// TIA Portal V20 export
FUNCTION_BLOCK "Sequence_2_AlignTable"   // FB243, LAD
AUTHOR : ERsystem_FA2_DH. Kim
// stored: IsIECCheckEnabled true, MemoryReserve 100, Namespace Unit1.Em4, SetENOAutomatically false
   VAR
      instSequenceLADStatus { ExternalWritable := 'False'} : "LAF_StatusLadSequence";
      instSequenceLADControl { ExternalWritable := 'False'} : "LAF_ControlLadSequence";
      statTonTime { ExternalWritable := 'False'} : Array[0..9999] of TON_TIME;
   END_VAR
   VAR_TEMP
      tempCustomerAction : Bool;   // Placeholder for possible actions
      tempDo_nothing_and_wait_for_init : Bool;   // Placeholder for doing nothing
      tempSafeStateCondition : Bool;   // Temp Condition for the equipment module to be in a safe state
   END_VAR
   VAR CONSTANT
      delayTime : Time := T#300ms;
      STEP_IDLE : DInt := 1;
      STEP_IMMEDIATE_STOP : DInt := 9001;   // Step executed when an immediate stop command is triggered for the sequence (i.e. when unit is in state aborting)
      JOB_1_STEP_01 : DInt := 101;
      JOB_1_STEP_10 : DInt := 110;
      JOB_1_STEP_20 : DInt := 120;
      JOB_1_STEP_30 : DInt := 130;
      JOB_1_STEP_40 : DInt := 140;
      JOB_1_STEP_41 : DInt := 141;
      JOB_1_STEP_42 : DInt := 142;
      JOB_1_STEP_50 : DInt := 150;
      JOB_1_STEP_51 : DInt := 151;
      JOB_1_STEP_52 : DInt := 152;
      JOB_1_STEP_60 : DInt := 160;
      JOB_1_STEP_61 : DInt := 161;
      JOB_1_STEP_62 : DInt := 162;
      JOB_1_STEP_70 : DInt := 170;
      JOB_1_STEP_80 : DInt := 180;
      JOB_1_STEP_81 : DInt := 181;
      JOB_1_STEP_90 : DInt := 190;
      JOB_2_STEP_01 : DInt := 201;
      JOB_2_STEP_10 : DInt := 210;
      JOB_2_STEP_20 : DInt := 220;
      JOB_2_STEP_30 : DInt := 230;
      JOB_2_STEP_90 : DInt := 290;
      JOB_3_STEP_01 : DInt := 301;
      JOB_3_STEP_10 : DInt := 310;
      JOB_3_STEP_20 : DInt := 320;
      JOB_3_STEP_80 : DInt := 380;
      JOB_3_STEP_90 : DInt := 390;
      JOB_4_STEP_01 : DInt := 401;
      JOB_4_STEP_10 : DInt := 410;
      JOB_4_STEP_11 : DInt := 411;
      JOB_4_STEP_20 : DInt := 420;
      JOB_4_STEP_21 : DInt := 421;
      JOB_4_STEP_30 : DInt := 430;
      JOB_4_STEP_80 : DInt := 480;
      JOB_4_STEP_81 : DInt := 481;
      JOB_4_STEP_90 : DInt := 490;
      JOB_22_STEP_01 : DInt := 2201;
      JOB_22_STEP_10 : DInt := 2210;
      JOB_22_STEP_20 : DInt := 2220;
      JOB_22_STEP_30 : DInt := 2230;
      JOB_22_STEP_40 : DInt := 2240;
      JOB_22_STEP_50 : DInt := 2250;
      JOB_22_STEP_80 : DInt := 2280;
      JOB_22_STEP_81 : DInt := 2281;
      JOB_22_STEP_90 : DInt := 2290;
      FALSE : Bool := FALSE;
      TRUE : Bool := TRUE;
   END_VAR
   VAR_TEMP   // added for the SCL form of the ladder/FBD networks
      _w1 : Bool;
   END_VAR
BEGIN

REGION Network 1: BLOCK INFO HEADER
   // (company) / (C) Copyright (year)
   // ---------------------------------------------------------------------------------
   // Title:                             (Title of this block)
   // Comment/Function: (that is implemented in the block)
   // Library/Family:           (that the source is dedicated to)
   // Author:                        (department / person in charge / contact)
   // Target System:          (test system with FW version)
   // Engineering:              TIA Portal (SW version)
   // Restrictions:               (OB types, etc.)
   // Requirements:           (hardware, technological package, etc.)
   // ---------------------------------------------------------------------------------
   // Change log table:
   // Version          | Date             | Signature      | Expert in charge  | Changes applied ------------------------|----------------------|-------------------------|--------------------------------|-----------------------
   // 001.000.000 | yyyy-mm-dd | 0x00000000 | (name of expert) | First released version
END_REGION

REGION Network 2: DESCRIPTION
   // This is a template block provided by the Automation Framework. It can be used to create an own project.
   // The Block Info Header is prepared to put in your own data.
   // Description of the block could be added here and the docu created by Code2Docu.
END_REGION

REGION Network 3: ******************** CONTROL ********************
END_REGION

REGION Network 4: Sequence Control
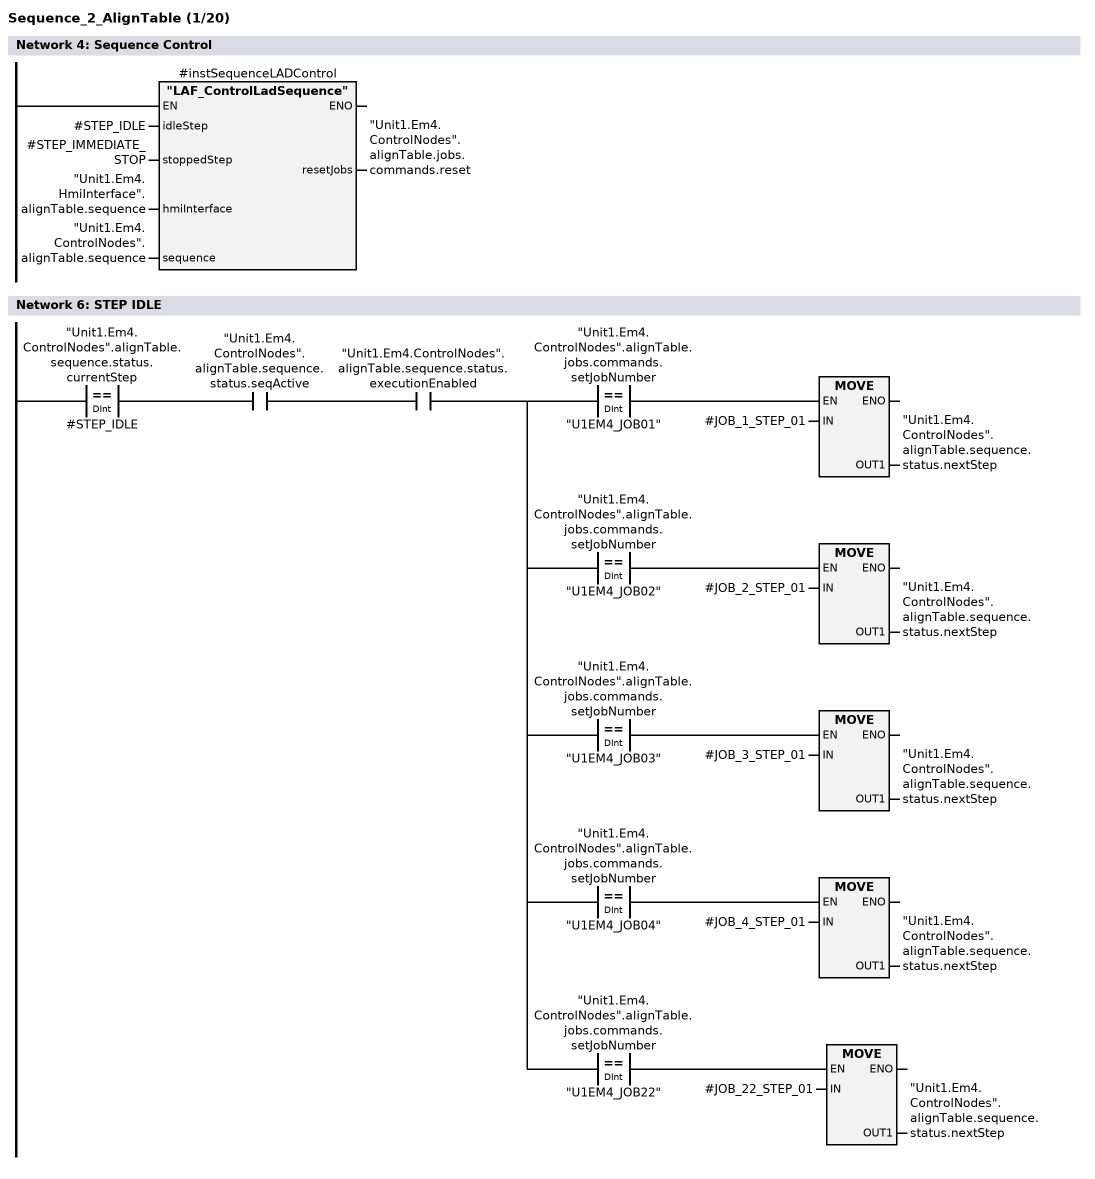
   RUNG wire#powerrail
      #instSequenceLADControl(idleStep := #STEP_IDLE, stoppedStep := #STEP_IMMEDIATE_STOP, hmiInterface := "Unit1.Em4.HmiInterface".alignTable.sequence, sequence := "Unit1.Em4.ControlNodes".alignTable.sequence, resetJobs => "Unit1.Em4.ControlNodes".alignTable.jobs.commands.reset)
   END_RUNG
   // the same network as SCL:
   #instSequenceLADControl(idleStep := #STEP_IDLE,   // "LAF_ControlLadSequence"
                           stoppedStep := #STEP_IMMEDIATE_STOP,
                           hmiInterface := "Unit1.Em4.HmiInterface".alignTable.sequence,
                           sequence := "Unit1.Em4.ControlNodes".alignTable.sequence,
                           resetJobs => "Unit1.Em4.ControlNodes".alignTable.jobs.commands.reset);
END_REGION

REGION Network 5: ******************** JOB SELECT ********************
END_REGION

REGION Network 6: STEP IDLE
   RUNG wire#powerrail
      { S7_Templates := "SrcType := DInt" } EQ_Contact(in1 := "Unit1.Em4.ControlNodes".alignTable.sequence.status.currentStep, in2 := #STEP_IDLE)
      Contact( "Unit1.Em4.ControlNodes".alignTable.sequence.status.seqActive )
      Contact( "Unit1.Em4.ControlNodes".alignTable.sequence.status.executionEnabled )
      wire#w1
      { S7_Templates := "SrcType := DInt" } EQ_Contact(in1 := "Unit1.Em4.ControlNodes".alignTable.jobs.commands.setJobNumber, in2 := "U1EM4_JOB01")
      Move(in := #JOB_1_STEP_01, out1 => "Unit1.Em4.ControlNodes".alignTable.sequence.status.nextStep)
   END_RUNG
   RUNG wire#w1
      { S7_Templates := "SrcType := DInt" } EQ_Contact(in1 := "Unit1.Em4.ControlNodes".alignTable.jobs.commands.setJobNumber, in2 := "U1EM4_JOB02")
      Move(in := #JOB_2_STEP_01, out1 => "Unit1.Em4.ControlNodes".alignTable.sequence.status.nextStep)
   END_RUNG
   RUNG wire#w1
      { S7_Templates := "SrcType := DInt" } EQ_Contact(in1 := "Unit1.Em4.ControlNodes".alignTable.jobs.commands.setJobNumber, in2 := "U1EM4_JOB03")
      Move(in := #JOB_3_STEP_01, out1 => "Unit1.Em4.ControlNodes".alignTable.sequence.status.nextStep)
   END_RUNG
   RUNG wire#w1
      { S7_Templates := "SrcType := DInt" } EQ_Contact(in1 := "Unit1.Em4.ControlNodes".alignTable.jobs.commands.setJobNumber, in2 := "U1EM4_JOB04")
      Move(in := #JOB_4_STEP_01, out1 => "Unit1.Em4.ControlNodes".alignTable.sequence.status.nextStep)
   END_RUNG
   RUNG wire#w1
      { S7_Templates := "SrcType := DInt" } EQ_Contact(in1 := "Unit1.Em4.ControlNodes".alignTable.jobs.commands.setJobNumber, in2 := "U1EM4_JOB22")
      Move(in := #JOB_22_STEP_01, out1 => "Unit1.Em4.ControlNodes".alignTable.sequence.status.nextStep)
   END_RUNG
   // the same network as SCL:
   #_w1 := ("Unit1.Em4.ControlNodes".alignTable.sequence.status.currentStep = #STEP_IDLE) AND "Unit1.Em4.ControlNodes".alignTable.sequence.status.seqActive AND "Unit1.Em4.ControlNodes".alignTable.sequence.status.executionEnabled;
   IF #_w1 AND ("Unit1.Em4.ControlNodes".alignTable.jobs.commands.setJobNumber = "U1EM4_JOB01") THEN
       "Unit1.Em4.ControlNodes".alignTable.sequence.status.nextStep := #JOB_1_STEP_01;
   END_IF;
   IF #_w1 AND ("Unit1.Em4.ControlNodes".alignTable.jobs.commands.setJobNumber = "U1EM4_JOB02") THEN
       "Unit1.Em4.ControlNodes".alignTable.sequence.status.nextStep := #JOB_2_STEP_01;
   END_IF;
   IF #_w1 AND ("Unit1.Em4.ControlNodes".alignTable.jobs.commands.setJobNumber = "U1EM4_JOB03") THEN
       "Unit1.Em4.ControlNodes".alignTable.sequence.status.nextStep := #JOB_3_STEP_01;
   END_IF;
   IF #_w1 AND ("Unit1.Em4.ControlNodes".alignTable.jobs.commands.setJobNumber = "U1EM4_JOB04") THEN
       "Unit1.Em4.ControlNodes".alignTable.sequence.status.nextStep := #JOB_4_STEP_01;
   END_IF;
   IF #_w1 AND ("Unit1.Em4.ControlNodes".alignTable.jobs.commands.setJobNumber = "U1EM4_JOB22") THEN
       "Unit1.Em4.ControlNodes".alignTable.sequence.status.nextStep := #JOB_22_STEP_01;
   END_IF;
END_REGION

REGION Network 7: ******************** JOB[1] EM HOMING ********************
END_REGION

REGION Network 8: Step[101] : JOB[1] Condition
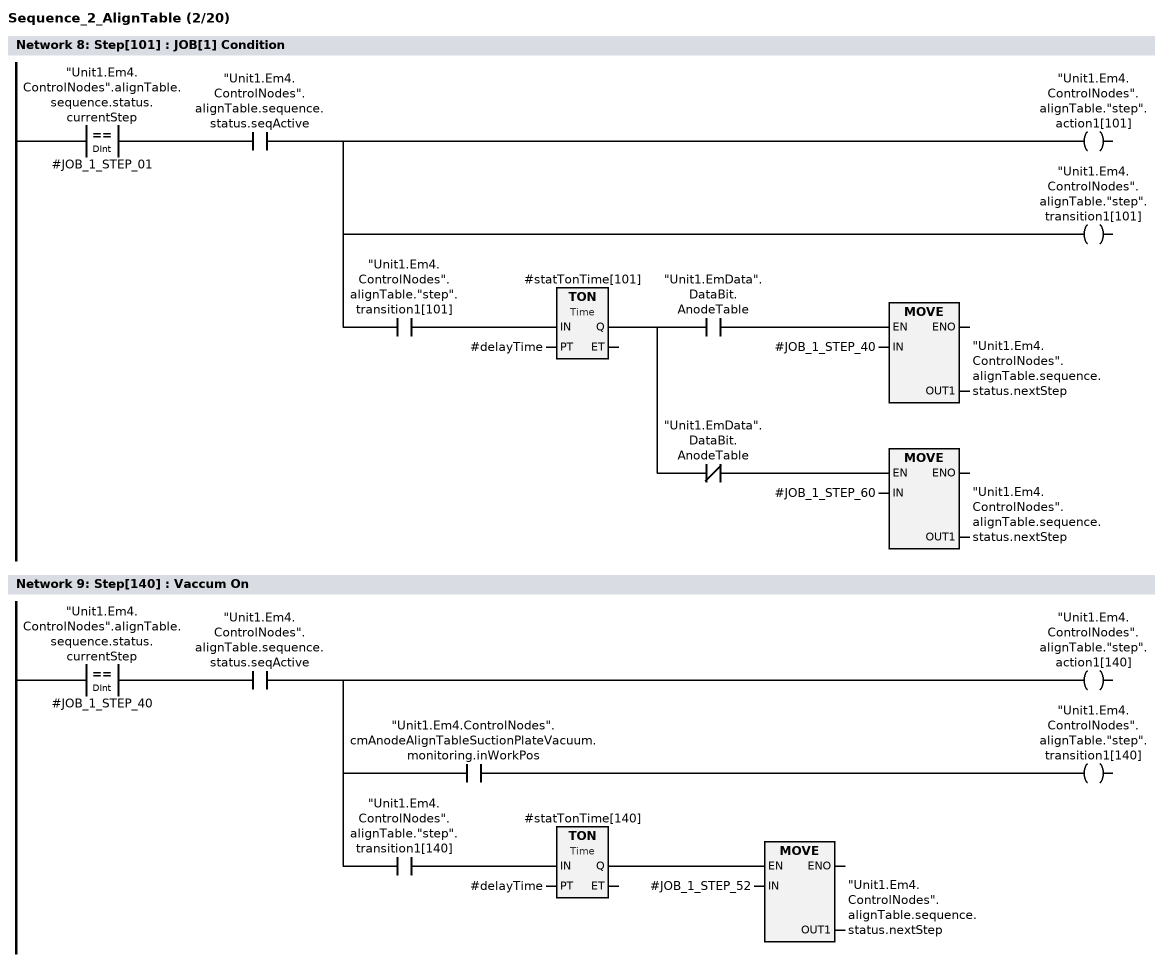
   RUNG wire#powerrail
      { S7_Templates := "SrcType := DInt" } EQ_Contact(in1 := "Unit1.Em4.ControlNodes".alignTable.sequence.status.currentStep, in2 := #JOB_1_STEP_01)
      Contact( "Unit1.Em4.ControlNodes".alignTable.sequence.status.seqActive )
      wire#w1
      Coil( "Unit1.Em4.ControlNodes".alignTable."step".action1[101] )
   END_RUNG
   RUNG wire#w1
      Coil( "Unit1.Em4.ControlNodes".alignTable."step".transition1[101] )
   END_RUNG
   RUNG wire#w1
      Contact( "Unit1.Em4.ControlNodes".alignTable."step".transition1[101] )
      { S7_Templates := "time_type := Time" } #statTonTime[101].TON(pt := #delayTime, et =>)
      wire#w2
      Contact( "Unit1.EmData".DataBit.AnodeTable )
      Move(in := #JOB_1_STEP_40, out1 => "Unit1.Em4.ControlNodes".alignTable.sequence.status.nextStep)
   END_RUNG
   RUNG wire#w2
      I_Contact( "Unit1.EmData".DataBit.AnodeTable )
      Move(in := #JOB_1_STEP_60, out1 => "Unit1.Em4.ControlNodes".alignTable.sequence.status.nextStep)
   END_RUNG
   // the same network as SCL:
   "Unit1.Em4.ControlNodes".alignTable."step".action1[101] := ("Unit1.Em4.ControlNodes".alignTable.sequence.status.currentStep = #JOB_1_STEP_01) AND "Unit1.Em4.ControlNodes".alignTable.sequence.status.seqActive;
   "Unit1.Em4.ControlNodes".alignTable."step".transition1[101] := ("Unit1.Em4.ControlNodes".alignTable.sequence.status.currentStep = #JOB_1_STEP_01) AND "Unit1.Em4.ControlNodes".alignTable.sequence.status.seqActive;
   #statTonTime[101].TON(IN := ("Unit1.Em4.ControlNodes".alignTable.sequence.status.currentStep = #JOB_1_STEP_01) AND "Unit1.Em4.ControlNodes".alignTable.sequence.status.seqActive AND "Unit1.Em4.ControlNodes".alignTable."step".transition1[101],
                         PT := #delayTime);
   IF #statTonTime[101].Q AND "Unit1.EmData".DataBit.AnodeTable THEN
       "Unit1.Em4.ControlNodes".alignTable.sequence.status.nextStep := #JOB_1_STEP_40;
   END_IF;
   IF #statTonTime[101].Q AND NOT "Unit1.EmData".DataBit.AnodeTable THEN
       "Unit1.Em4.ControlNodes".alignTable.sequence.status.nextStep := #JOB_1_STEP_60;
   END_IF;
END_REGION

REGION Network 9: Step[140] : Vaccum On
   RUNG wire#powerrail
      { S7_Templates := "SrcType := DInt" } EQ_Contact(in1 := "Unit1.Em4.ControlNodes".alignTable.sequence.status.currentStep, in2 := #JOB_1_STEP_40)
      Contact( "Unit1.Em4.ControlNodes".alignTable.sequence.status.seqActive )
      wire#w1
      Coil( "Unit1.Em4.ControlNodes".alignTable."step".action1[140] )
   END_RUNG
   RUNG wire#w1
      Contact( "Unit1.Em4.ControlNodes".cmAnodeAlignTableSuctionPlateVacuum.monitoring.inWorkPos )
      Coil( "Unit1.Em4.ControlNodes".alignTable."step".transition1[140] )
   END_RUNG
   RUNG wire#w1
      Contact( "Unit1.Em4.ControlNodes".alignTable."step".transition1[140] )
      { S7_Templates := "time_type := Time" } #statTonTime[140].TON(pt := #delayTime, et =>)
      Move(in := #JOB_1_STEP_52, out1 => "Unit1.Em4.ControlNodes".alignTable.sequence.status.nextStep)
   END_RUNG
   // the same network as SCL:
   "Unit1.Em4.ControlNodes".alignTable."step".action1[140] := ("Unit1.Em4.ControlNodes".alignTable.sequence.status.currentStep = #JOB_1_STEP_40) AND "Unit1.Em4.ControlNodes".alignTable.sequence.status.seqActive;
   "Unit1.Em4.ControlNodes".alignTable."step".transition1[140] := ("Unit1.Em4.ControlNodes".alignTable.sequence.status.currentStep = #JOB_1_STEP_40) AND "Unit1.Em4.ControlNodes".alignTable.sequence.status.seqActive AND "Unit1.Em4.ControlNodes".cmAnodeAlignTableSuctionPlateVacuum.monitoring.inWorkPos;
   #statTonTime[140].TON(IN := ("Unit1.Em4.ControlNodes".alignTable.sequence.status.currentStep = #JOB_1_STEP_40) AND "Unit1.Em4.ControlNodes".alignTable.sequence.status.seqActive AND "Unit1.Em4.ControlNodes".alignTable."step".transition1[140],
                         PT := #delayTime);
   IF #statTonTime[140].Q THEN
       "Unit1.Em4.ControlNodes".alignTable.sequence.status.nextStep := #JOB_1_STEP_52;
   END_IF;
END_REGION

REGION Network 10: Step[141] : Align Table → Main P&P [Load Done]
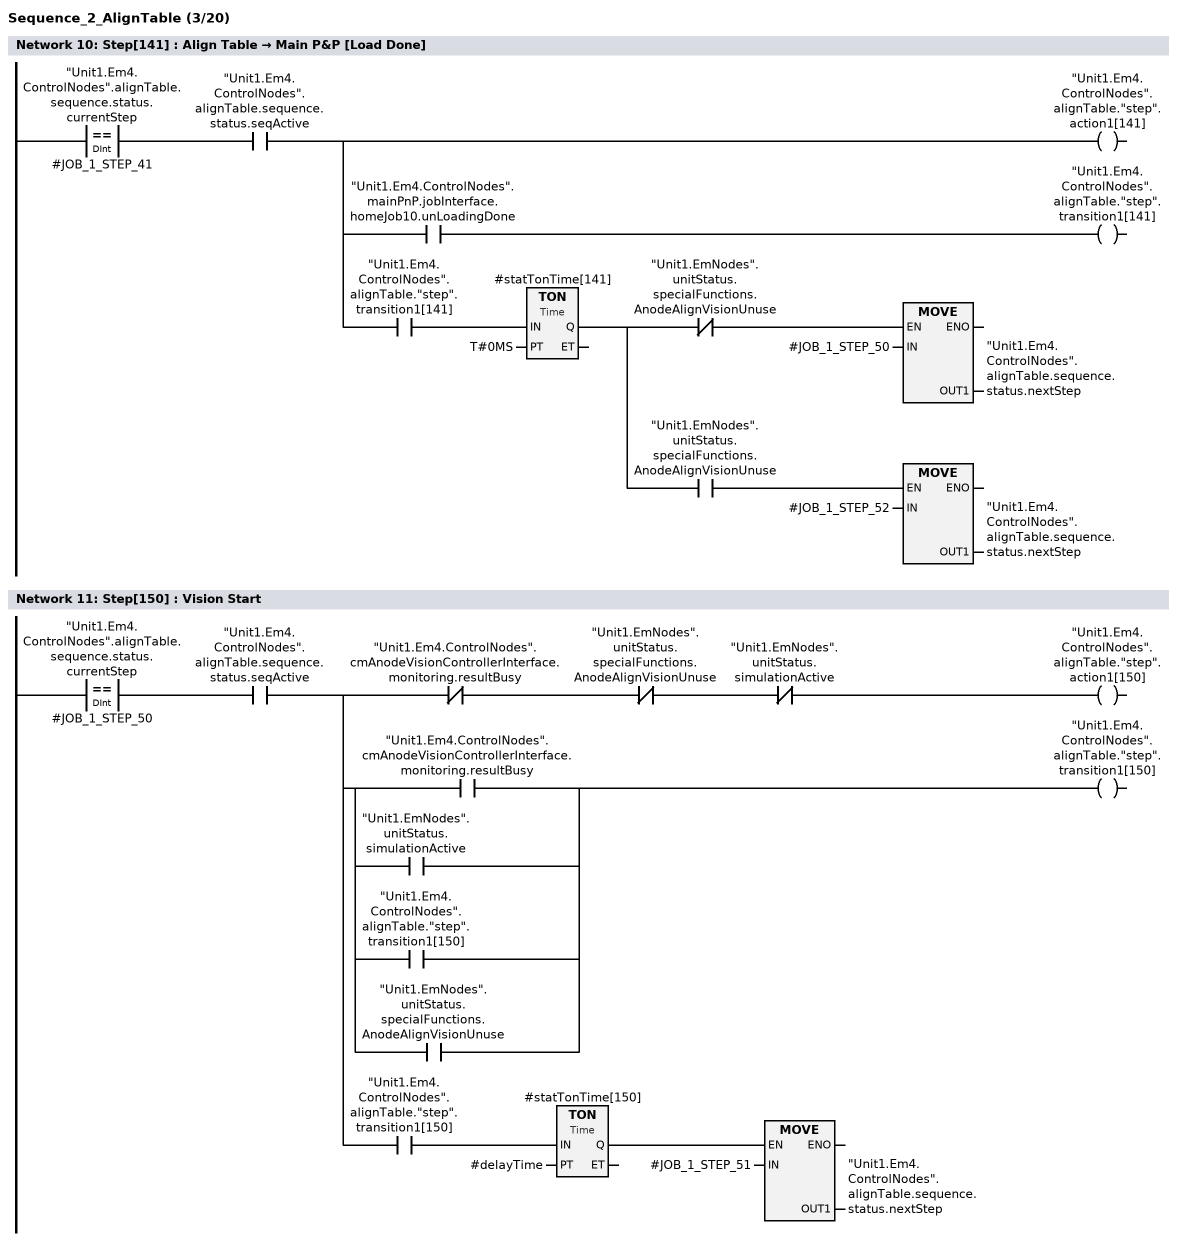
   RUNG wire#powerrail
      { S7_Templates := "SrcType := DInt" } EQ_Contact(in1 := "Unit1.Em4.ControlNodes".alignTable.sequence.status.currentStep, in2 := #JOB_1_STEP_41)
      Contact( "Unit1.Em4.ControlNodes".alignTable.sequence.status.seqActive )
      wire#w1
      Coil( "Unit1.Em4.ControlNodes".alignTable."step".action1[141] )
   END_RUNG
   RUNG wire#w1
      Contact( "Unit1.Em4.ControlNodes".mainPnP.jobInterface.homeJob10.unLoadingDone )
      Coil( "Unit1.Em4.ControlNodes".alignTable."step".transition1[141] )
   END_RUNG
   RUNG wire#w1
      Contact( "Unit1.Em4.ControlNodes".alignTable."step".transition1[141] )
      { S7_Templates := "time_type := Time" } #statTonTime[141].TON(pt := T#0MS, et =>)
      wire#w2
      I_Contact( "Unit1.EmNodes".unitStatus.specialFunctions.AnodeAlignVisionUnuse )
      Move(in := #JOB_1_STEP_50, out1 => "Unit1.Em4.ControlNodes".alignTable.sequence.status.nextStep)
   END_RUNG
   RUNG wire#w2
      Contact( "Unit1.EmNodes".unitStatus.specialFunctions.AnodeAlignVisionUnuse )
      Move(in := #JOB_1_STEP_52, out1 => "Unit1.Em4.ControlNodes".alignTable.sequence.status.nextStep)
   END_RUNG
   // the same network as SCL:
   "Unit1.Em4.ControlNodes".alignTable."step".action1[141] := ("Unit1.Em4.ControlNodes".alignTable.sequence.status.currentStep = #JOB_1_STEP_41) AND "Unit1.Em4.ControlNodes".alignTable.sequence.status.seqActive;
   "Unit1.Em4.ControlNodes".alignTable."step".transition1[141] := ("Unit1.Em4.ControlNodes".alignTable.sequence.status.currentStep = #JOB_1_STEP_41) AND "Unit1.Em4.ControlNodes".alignTable.sequence.status.seqActive AND "Unit1.Em4.ControlNodes".mainPnP.jobInterface.homeJob10.unLoadingDone;
   #statTonTime[141].TON(IN := ("Unit1.Em4.ControlNodes".alignTable.sequence.status.currentStep = #JOB_1_STEP_41) AND "Unit1.Em4.ControlNodes".alignTable.sequence.status.seqActive AND "Unit1.Em4.ControlNodes".alignTable."step".transition1[141],
                         PT := T#0MS);
   IF #statTonTime[141].Q AND NOT "Unit1.EmNodes".unitStatus.specialFunctions.AnodeAlignVisionUnuse THEN
       "Unit1.Em4.ControlNodes".alignTable.sequence.status.nextStep := #JOB_1_STEP_50;
   END_IF;
   IF #statTonTime[141].Q AND "Unit1.EmNodes".unitStatus.specialFunctions.AnodeAlignVisionUnuse THEN
       "Unit1.Em4.ControlNodes".alignTable.sequence.status.nextStep := #JOB_1_STEP_52;
   END_IF;
END_REGION

REGION Network 11: Step[150] : Vision Start
   RUNG wire#powerrail
      { S7_Templates := "SrcType := DInt" } EQ_Contact(in1 := "Unit1.Em4.ControlNodes".alignTable.sequence.status.currentStep, in2 := #JOB_1_STEP_50)
      Contact( "Unit1.Em4.ControlNodes".alignTable.sequence.status.seqActive )
      wire#w1
      I_Contact( "Unit1.Em4.ControlNodes".cmAnodeVisionControllerInterface.monitoring.resultBusy )
      I_Contact( "Unit1.EmNodes".unitStatus.specialFunctions.AnodeAlignVisionUnuse )
      I_Contact( "Unit1.EmNodes".unitStatus.simulationActive )
      Coil( "Unit1.Em4.ControlNodes".alignTable."step".action1[150] )
   END_RUNG
   RUNG wire#w1
      Contact( "Unit1.Em4.ControlNodes".cmAnodeVisionControllerInterface.monitoring.resultBusy )
      wire#w2
      Coil( "Unit1.Em4.ControlNodes".alignTable."step".transition1[150] )
   END_RUNG
   RUNG wire#w1
      Contact( "Unit1.EmNodes".unitStatus.simulationActive )
   END_RUNG wire#w2
   RUNG wire#w1
      Contact( "Unit1.Em4.ControlNodes".alignTable."step".transition1[150] )
   END_RUNG wire#w2
   RUNG wire#w1
      Contact( "Unit1.EmNodes".unitStatus.specialFunctions.AnodeAlignVisionUnuse )
   END_RUNG wire#w2
   RUNG wire#w1
      Contact( "Unit1.Em4.ControlNodes".alignTable."step".transition1[150] )
      { S7_Templates := "time_type := Time" } #statTonTime[150].TON(pt := #delayTime, et =>)
      Move(in := #JOB_1_STEP_51, out1 => "Unit1.Em4.ControlNodes".alignTable.sequence.status.nextStep)
   END_RUNG
   // the same network as SCL:
   #_w1 := ("Unit1.Em4.ControlNodes".alignTable.sequence.status.currentStep = #JOB_1_STEP_50) AND "Unit1.Em4.ControlNodes".alignTable.sequence.status.seqActive;
   "Unit1.Em4.ControlNodes".alignTable."step".action1[150] := #_w1 AND NOT "Unit1.Em4.ControlNodes".cmAnodeVisionControllerInterface.monitoring.resultBusy AND NOT "Unit1.EmNodes".unitStatus.specialFunctions.AnodeAlignVisionUnuse AND NOT "Unit1.EmNodes".unitStatus.simulationActive;
   "Unit1.Em4.ControlNodes".alignTable."step".transition1[150] := #_w1 AND ("Unit1.Em4.ControlNodes".cmAnodeVisionControllerInterface.monitoring.resultBusy OR "Unit1.EmNodes".unitStatus.simulationActive OR "Unit1.Em4.ControlNodes".alignTable."step".transition1[150] OR "Unit1.EmNodes".unitStatus.specialFunctions.AnodeAlignVisionUnuse);
   #statTonTime[150].TON(IN := #_w1 AND "Unit1.Em4.ControlNodes".alignTable."step".transition1[150],
                         PT := #delayTime);
   IF #statTonTime[150].Q THEN
       "Unit1.Em4.ControlNodes".alignTable.sequence.status.nextStep := #JOB_1_STEP_51;
   END_IF;
END_REGION

REGION Network 12: Step[151] : Vision Result
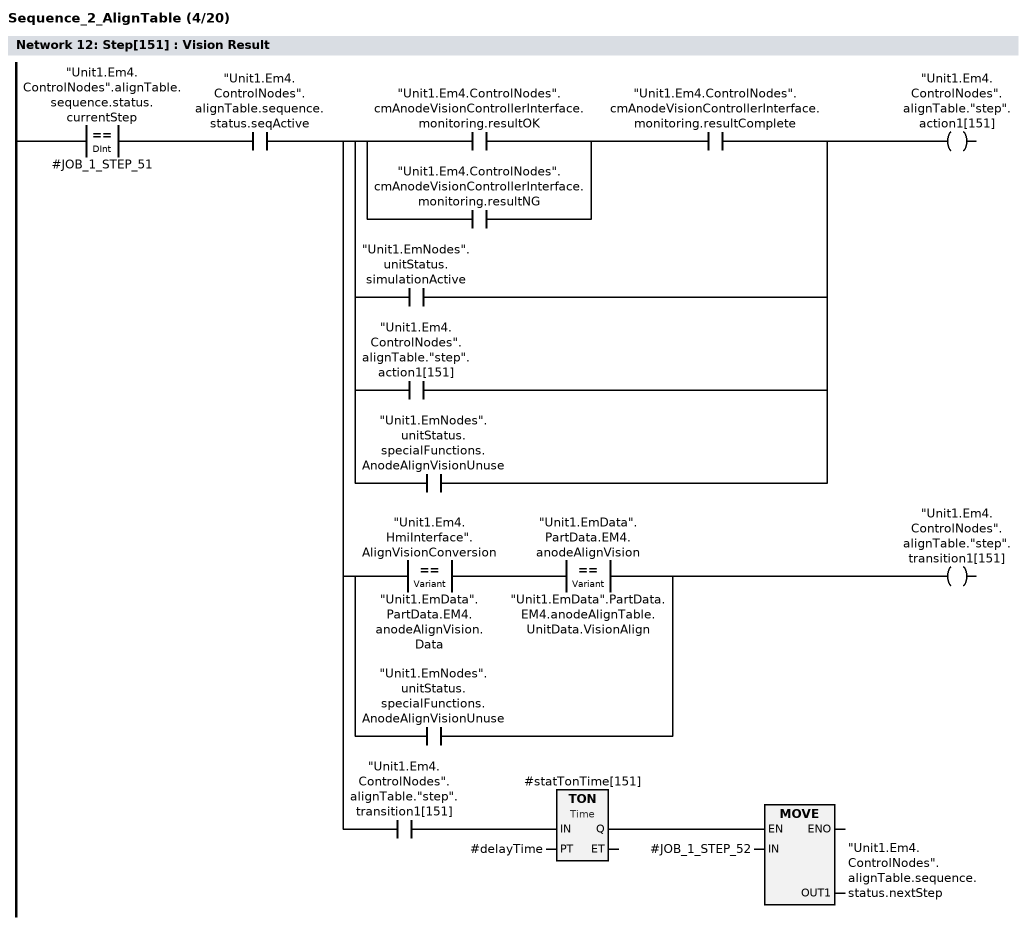
   RUNG wire#powerrail
      { S7_Templates := "SrcType := DInt" } EQ_Contact(in1 := "Unit1.Em4.ControlNodes".alignTable.sequence.status.currentStep, in2 := #JOB_1_STEP_51)
      Contact( "Unit1.Em4.ControlNodes".alignTable.sequence.status.seqActive )
      wire#w1
      Contact( "Unit1.Em4.ControlNodes".cmAnodeVisionControllerInterface.monitoring.resultOK )
      wire#w2
      Contact( "Unit1.Em4.ControlNodes".cmAnodeVisionControllerInterface.monitoring.resultComplete )
      wire#w3
      Coil( "Unit1.Em4.ControlNodes".alignTable."step".action1[151] )
   END_RUNG
   RUNG wire#w1
      Contact( "Unit1.Em4.ControlNodes".cmAnodeVisionControllerInterface.monitoring.resultNG )
   END_RUNG wire#w2
   RUNG wire#w1
      Contact( "Unit1.EmNodes".unitStatus.simulationActive )
   END_RUNG wire#w3
   RUNG wire#w1
      Contact( "Unit1.Em4.ControlNodes".alignTable."step".action1[151] )
   END_RUNG wire#w3
   RUNG wire#w1
      Contact( "Unit1.EmNodes".unitStatus.specialFunctions.AnodeAlignVisionUnuse )
   END_RUNG wire#w3
   RUNG wire#w1
      { S7_Templates := "SrcType := Variant" } EQ_Contact(in1 := "Unit1.Em4.HmiInterface".AlignVisionConversion, in2 := "Unit1.EmData".PartData.EM4.anodeAlignVision.Data)
      { S7_Templates := "SrcType := Variant" } EQ_Contact(in1 := "Unit1.EmData".PartData.EM4.anodeAlignVision, in2 := "Unit1.EmData".PartData.EM4.anodeAlignTable.UnitData.VisionAlign)
      wire#w4
      Coil( "Unit1.Em4.ControlNodes".alignTable."step".transition1[151] )
   END_RUNG
   RUNG wire#w1
      Contact( "Unit1.EmNodes".unitStatus.specialFunctions.AnodeAlignVisionUnuse )
   END_RUNG wire#w4
   RUNG wire#w1
      Contact( "Unit1.Em4.ControlNodes".alignTable."step".transition1[151] )
      { S7_Templates := "time_type := Time" } #statTonTime[151].TON(pt := #delayTime, et =>)
      Move(in := #JOB_1_STEP_52, out1 => "Unit1.Em4.ControlNodes".alignTable.sequence.status.nextStep)
   END_RUNG
   // the same network as SCL:
   #_w1 := ("Unit1.Em4.ControlNodes".alignTable.sequence.status.currentStep = #JOB_1_STEP_51) AND "Unit1.Em4.ControlNodes".alignTable.sequence.status.seqActive;
   "Unit1.Em4.ControlNodes".alignTable."step".action1[151] := #_w1 AND ((("Unit1.Em4.ControlNodes".cmAnodeVisionControllerInterface.monitoring.resultOK OR "Unit1.Em4.ControlNodes".cmAnodeVisionControllerInterface.monitoring.resultNG) AND "Unit1.Em4.ControlNodes".cmAnodeVisionControllerInterface.monitoring.resultComplete) OR "Unit1.EmNodes".unitStatus.simulationActive OR "Unit1.Em4.ControlNodes".alignTable."step".action1[151] OR "Unit1.EmNodes".unitStatus.specialFunctions.AnodeAlignVisionUnuse);
   "Unit1.Em4.ControlNodes".alignTable."step".transition1[151] := #_w1 AND ((("Unit1.Em4.HmiInterface".AlignVisionConversion = "Unit1.EmData".PartData.EM4.anodeAlignVision.Data) AND ("Unit1.EmData".PartData.EM4.anodeAlignVision = "Unit1.EmData".PartData.EM4.anodeAlignTable.UnitData.VisionAlign)) OR "Unit1.EmNodes".unitStatus.specialFunctions.AnodeAlignVisionUnuse);
   #statTonTime[151].TON(IN := #_w1 AND "Unit1.Em4.ControlNodes".alignTable."step".transition1[151],
                         PT := #delayTime);
   IF #statTonTime[151].Q THEN
       "Unit1.Em4.ControlNodes".alignTable.sequence.status.nextStep := #JOB_1_STEP_52;
   END_IF;
END_REGION

REGION Network 13: Step[152] : Align Table X,Y1,Y2-Axis Work Pos
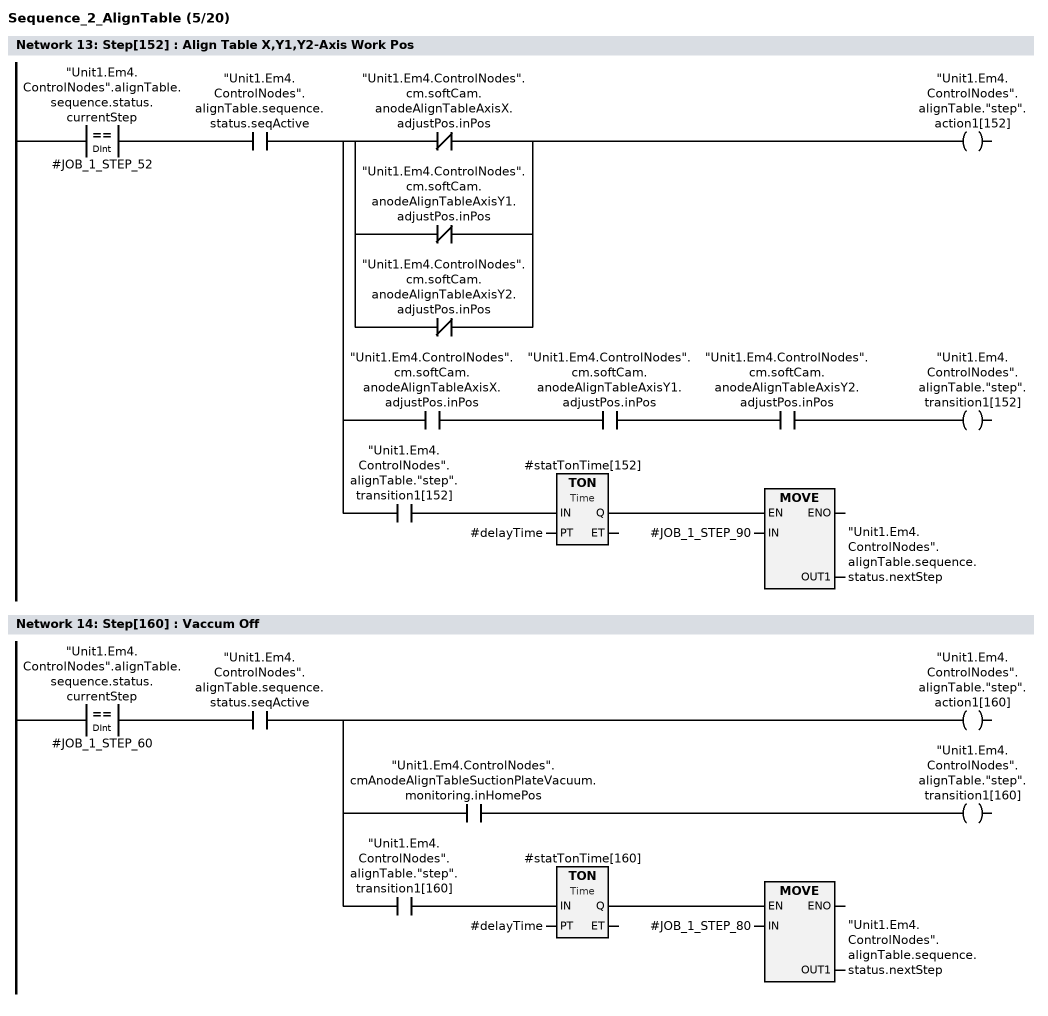
   RUNG wire#powerrail
      { S7_Templates := "SrcType := DInt" } EQ_Contact(in1 := "Unit1.Em4.ControlNodes".alignTable.sequence.status.currentStep, in2 := #JOB_1_STEP_52)
      Contact( "Unit1.Em4.ControlNodes".alignTable.sequence.status.seqActive )
      wire#w1
      I_Contact( "Unit1.Em4.ControlNodes".cm.softCam.anodeAlignTableAxisX.adjustPos.inPos )
      wire#w2
      Coil( "Unit1.Em4.ControlNodes".alignTable."step".action1[152] )
   END_RUNG
   RUNG wire#w1
      I_Contact( "Unit1.Em4.ControlNodes".cm.softCam.anodeAlignTableAxisY1.adjustPos.inPos )
   END_RUNG wire#w2
   RUNG wire#w1
      I_Contact( "Unit1.Em4.ControlNodes".cm.softCam.anodeAlignTableAxisY2.adjustPos.inPos )
   END_RUNG wire#w2
   RUNG wire#w1
      Contact( "Unit1.Em4.ControlNodes".cm.softCam.anodeAlignTableAxisX.adjustPos.inPos )
      Contact( "Unit1.Em4.ControlNodes".cm.softCam.anodeAlignTableAxisY1.adjustPos.inPos )
      Contact( "Unit1.Em4.ControlNodes".cm.softCam.anodeAlignTableAxisY2.adjustPos.inPos )
      Coil( "Unit1.Em4.ControlNodes".alignTable."step".transition1[152] )
   END_RUNG
   RUNG wire#w1
      Contact( "Unit1.Em4.ControlNodes".alignTable."step".transition1[152] )
      { S7_Templates := "time_type := Time" } #statTonTime[152].TON(pt := #delayTime, et =>)
      Move(in := #JOB_1_STEP_90, out1 => "Unit1.Em4.ControlNodes".alignTable.sequence.status.nextStep)
   END_RUNG
   // the same network as SCL:
   #_w1 := ("Unit1.Em4.ControlNodes".alignTable.sequence.status.currentStep = #JOB_1_STEP_52) AND "Unit1.Em4.ControlNodes".alignTable.sequence.status.seqActive;
   "Unit1.Em4.ControlNodes".alignTable."step".action1[152] := #_w1 AND (NOT "Unit1.Em4.ControlNodes".cm.softCam.anodeAlignTableAxisX.adjustPos.inPos OR NOT "Unit1.Em4.ControlNodes".cm.softCam.anodeAlignTableAxisY1.adjustPos.inPos OR NOT "Unit1.Em4.ControlNodes".cm.softCam.anodeAlignTableAxisY2.adjustPos.inPos);
   "Unit1.Em4.ControlNodes".alignTable."step".transition1[152] := #_w1 AND "Unit1.Em4.ControlNodes".cm.softCam.anodeAlignTableAxisX.adjustPos.inPos AND "Unit1.Em4.ControlNodes".cm.softCam.anodeAlignTableAxisY1.adjustPos.inPos AND "Unit1.Em4.ControlNodes".cm.softCam.anodeAlignTableAxisY2.adjustPos.inPos;
   #statTonTime[152].TON(IN := #_w1 AND "Unit1.Em4.ControlNodes".alignTable."step".transition1[152],
                         PT := #delayTime);
   IF #statTonTime[152].Q THEN
       "Unit1.Em4.ControlNodes".alignTable.sequence.status.nextStep := #JOB_1_STEP_90;
   END_IF;
END_REGION

REGION Network 14: Step[160] : Vaccum Off
   RUNG wire#powerrail
      { S7_Templates := "SrcType := DInt" } EQ_Contact(in1 := "Unit1.Em4.ControlNodes".alignTable.sequence.status.currentStep, in2 := #JOB_1_STEP_60)
      Contact( "Unit1.Em4.ControlNodes".alignTable.sequence.status.seqActive )
      wire#w1
      Coil( "Unit1.Em4.ControlNodes".alignTable."step".action1[160] )
   END_RUNG
   RUNG wire#w1
      Contact( "Unit1.Em4.ControlNodes".cmAnodeAlignTableSuctionPlateVacuum.monitoring.inHomePos )
      Coil( "Unit1.Em4.ControlNodes".alignTable."step".transition1[160] )
   END_RUNG
   RUNG wire#w1
      Contact( "Unit1.Em4.ControlNodes".alignTable."step".transition1[160] )
      { S7_Templates := "time_type := Time" } #statTonTime[160].TON(pt := #delayTime, et =>)
      Move(in := #JOB_1_STEP_80, out1 => "Unit1.Em4.ControlNodes".alignTable.sequence.status.nextStep)
   END_RUNG
   // the same network as SCL:
   "Unit1.Em4.ControlNodes".alignTable."step".action1[160] := ("Unit1.Em4.ControlNodes".alignTable.sequence.status.currentStep = #JOB_1_STEP_60) AND "Unit1.Em4.ControlNodes".alignTable.sequence.status.seqActive;
   "Unit1.Em4.ControlNodes".alignTable."step".transition1[160] := ("Unit1.Em4.ControlNodes".alignTable.sequence.status.currentStep = #JOB_1_STEP_60) AND "Unit1.Em4.ControlNodes".alignTable.sequence.status.seqActive AND "Unit1.Em4.ControlNodes".cmAnodeAlignTableSuctionPlateVacuum.monitoring.inHomePos;
   #statTonTime[160].TON(IN := ("Unit1.Em4.ControlNodes".alignTable.sequence.status.currentStep = #JOB_1_STEP_60) AND "Unit1.Em4.ControlNodes".alignTable.sequence.status.seqActive AND "Unit1.Em4.ControlNodes".alignTable."step".transition1[160],
                         PT := #delayTime);
   IF #statTonTime[160].Q THEN
       "Unit1.Em4.ControlNodes".alignTable.sequence.status.nextStep := #JOB_1_STEP_80;
   END_IF;
END_REGION

REGION Network 15: Step[161] : Align Table → Main P&P [Unload Done]
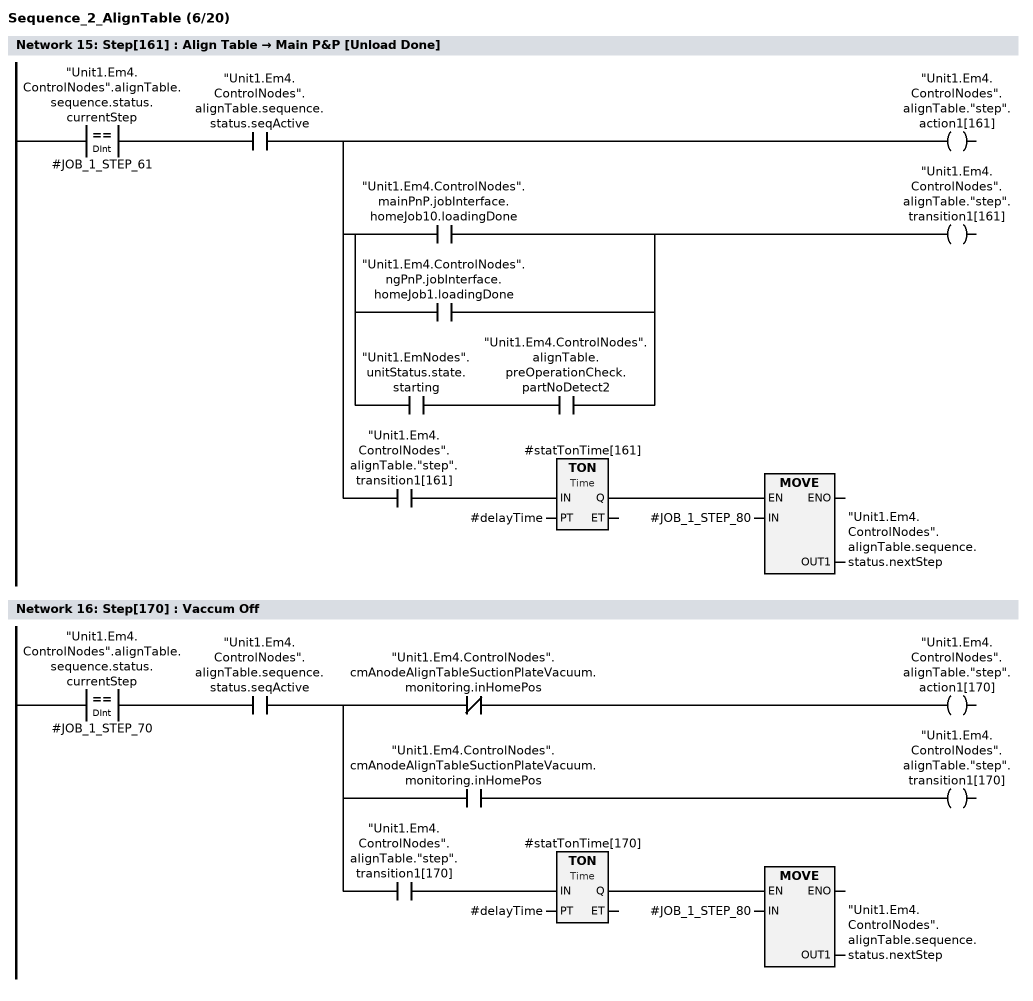
   RUNG wire#powerrail
      { S7_Templates := "SrcType := DInt" } EQ_Contact(in1 := "Unit1.Em4.ControlNodes".alignTable.sequence.status.currentStep, in2 := #JOB_1_STEP_61)
      Contact( "Unit1.Em4.ControlNodes".alignTable.sequence.status.seqActive )
      wire#w1
      Coil( "Unit1.Em4.ControlNodes".alignTable."step".action1[161] )
   END_RUNG
   RUNG wire#w1
      Contact( "Unit1.Em4.ControlNodes".mainPnP.jobInterface.homeJob10.loadingDone )
      wire#w2
      Coil( "Unit1.Em4.ControlNodes".alignTable."step".transition1[161] )
   END_RUNG
   RUNG wire#w1
      Contact( "Unit1.Em4.ControlNodes".ngPnP.jobInterface.homeJob1.loadingDone )
   END_RUNG wire#w2
   RUNG wire#w1
      Contact( "Unit1.EmNodes".unitStatus.state.starting )
      Contact( "Unit1.Em4.ControlNodes".alignTable.preOperationCheck.partNoDetect2 )
   END_RUNG wire#w2
   RUNG wire#w1
      Contact( "Unit1.Em4.ControlNodes".alignTable."step".transition1[161] )
      { S7_Templates := "time_type := Time" } #statTonTime[161].TON(pt := #delayTime, et =>)
      Move(in := #JOB_1_STEP_80, out1 => "Unit1.Em4.ControlNodes".alignTable.sequence.status.nextStep)
   END_RUNG
   // the same network as SCL:
   "Unit1.Em4.ControlNodes".alignTable."step".action1[161] := ("Unit1.Em4.ControlNodes".alignTable.sequence.status.currentStep = #JOB_1_STEP_61) AND "Unit1.Em4.ControlNodes".alignTable.sequence.status.seqActive;
   "Unit1.Em4.ControlNodes".alignTable."step".transition1[161] := ("Unit1.Em4.ControlNodes".alignTable.sequence.status.currentStep = #JOB_1_STEP_61) AND "Unit1.Em4.ControlNodes".alignTable.sequence.status.seqActive AND ("Unit1.Em4.ControlNodes".mainPnP.jobInterface.homeJob10.loadingDone OR "Unit1.Em4.ControlNodes".ngPnP.jobInterface.homeJob1.loadingDone OR ("Unit1.EmNodes".unitStatus.state.starting AND "Unit1.Em4.ControlNodes".alignTable.preOperationCheck.partNoDetect2));
   #statTonTime[161].TON(IN := ("Unit1.Em4.ControlNodes".alignTable.sequence.status.currentStep = #JOB_1_STEP_61) AND "Unit1.Em4.ControlNodes".alignTable.sequence.status.seqActive AND "Unit1.Em4.ControlNodes".alignTable."step".transition1[161],
                         PT := #delayTime);
   IF #statTonTime[161].Q THEN
       "Unit1.Em4.ControlNodes".alignTable.sequence.status.nextStep := #JOB_1_STEP_80;
   END_IF;
END_REGION

REGION Network 16: Step[170] : Vaccum Off
   RUNG wire#powerrail
      { S7_Templates := "SrcType := DInt" } EQ_Contact(in1 := "Unit1.Em4.ControlNodes".alignTable.sequence.status.currentStep, in2 := #JOB_1_STEP_70)
      Contact( "Unit1.Em4.ControlNodes".alignTable.sequence.status.seqActive )
      wire#w1
      I_Contact( "Unit1.Em4.ControlNodes".cmAnodeAlignTableSuctionPlateVacuum.monitoring.inHomePos )
      Coil( "Unit1.Em4.ControlNodes".alignTable."step".action1[170] )
   END_RUNG
   RUNG wire#w1
      Contact( "Unit1.Em4.ControlNodes".cmAnodeAlignTableSuctionPlateVacuum.monitoring.inHomePos )
      Coil( "Unit1.Em4.ControlNodes".alignTable."step".transition1[170] )
   END_RUNG
   RUNG wire#w1
      Contact( "Unit1.Em4.ControlNodes".alignTable."step".transition1[170] )
      { S7_Templates := "time_type := Time" } #statTonTime[170].TON(pt := #delayTime, et =>)
      Move(in := #JOB_1_STEP_80, out1 => "Unit1.Em4.ControlNodes".alignTable.sequence.status.nextStep)
   END_RUNG
   // the same network as SCL:
   #_w1 := ("Unit1.Em4.ControlNodes".alignTable.sequence.status.currentStep = #JOB_1_STEP_70) AND "Unit1.Em4.ControlNodes".alignTable.sequence.status.seqActive;
   "Unit1.Em4.ControlNodes".alignTable."step".action1[170] := #_w1 AND NOT "Unit1.Em4.ControlNodes".cmAnodeAlignTableSuctionPlateVacuum.monitoring.inHomePos;
   "Unit1.Em4.ControlNodes".alignTable."step".transition1[170] := #_w1 AND "Unit1.Em4.ControlNodes".cmAnodeAlignTableSuctionPlateVacuum.monitoring.inHomePos;
   #statTonTime[170].TON(IN := #_w1 AND "Unit1.Em4.ControlNodes".alignTable."step".transition1[170],
                         PT := #delayTime);
   IF #statTonTime[170].Q THEN
       "Unit1.Em4.ControlNodes".alignTable.sequence.status.nextStep := #JOB_1_STEP_80;
   END_IF;
END_REGION

REGION Network 17: Step[180] : Align Table X,Y1,Y2-Axis Wait Pos
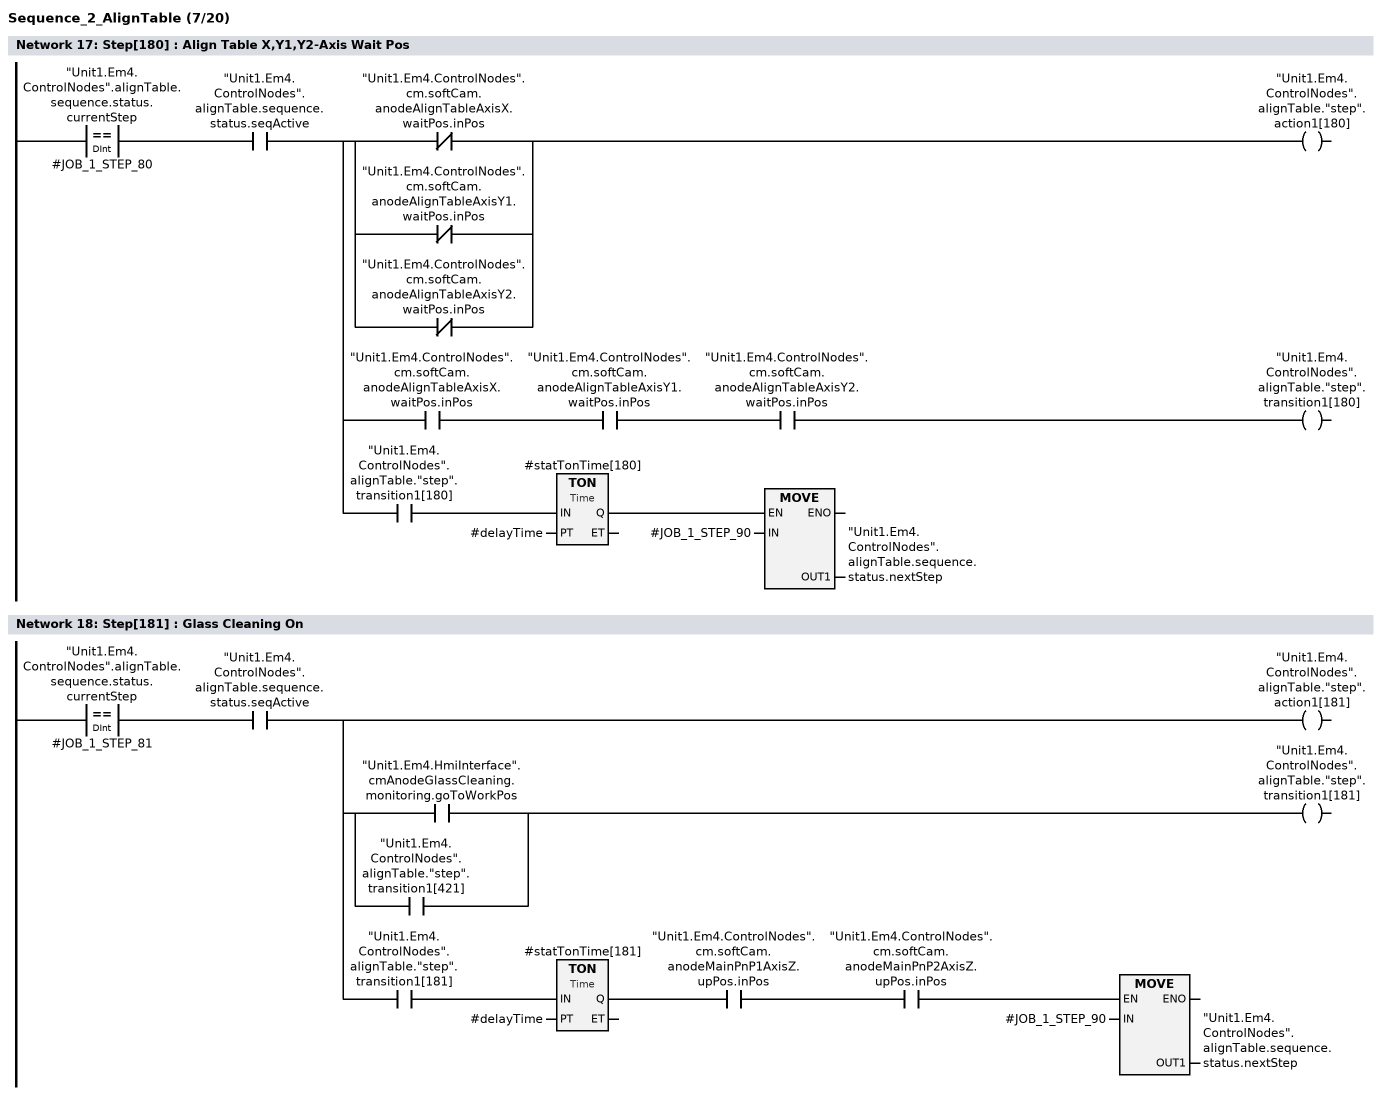
   RUNG wire#powerrail
      { S7_Templates := "SrcType := DInt" } EQ_Contact(in1 := "Unit1.Em4.ControlNodes".alignTable.sequence.status.currentStep, in2 := #JOB_1_STEP_80)
      Contact( "Unit1.Em4.ControlNodes".alignTable.sequence.status.seqActive )
      wire#w1
      I_Contact( "Unit1.Em4.ControlNodes".cm.softCam.anodeAlignTableAxisX.waitPos.inPos )
      wire#w2
      Coil( "Unit1.Em4.ControlNodes".alignTable."step".action1[180] )
   END_RUNG
   RUNG wire#w1
      I_Contact( "Unit1.Em4.ControlNodes".cm.softCam.anodeAlignTableAxisY1.waitPos.inPos )
   END_RUNG wire#w2
   RUNG wire#w1
      I_Contact( "Unit1.Em4.ControlNodes".cm.softCam.anodeAlignTableAxisY2.waitPos.inPos )
   END_RUNG wire#w2
   RUNG wire#w1
      Contact( "Unit1.Em4.ControlNodes".cm.softCam.anodeAlignTableAxisX.waitPos.inPos )
      Contact( "Unit1.Em4.ControlNodes".cm.softCam.anodeAlignTableAxisY1.waitPos.inPos )
      Contact( "Unit1.Em4.ControlNodes".cm.softCam.anodeAlignTableAxisY2.waitPos.inPos )
      Coil( "Unit1.Em4.ControlNodes".alignTable."step".transition1[180] )
   END_RUNG
   RUNG wire#w1
      Contact( "Unit1.Em4.ControlNodes".alignTable."step".transition1[180] )
      { S7_Templates := "time_type := Time" } #statTonTime[180].TON(pt := #delayTime, et =>)
      Move(in := #JOB_1_STEP_90, out1 => "Unit1.Em4.ControlNodes".alignTable.sequence.status.nextStep)
   END_RUNG
   // the same network as SCL:
   #_w1 := ("Unit1.Em4.ControlNodes".alignTable.sequence.status.currentStep = #JOB_1_STEP_80) AND "Unit1.Em4.ControlNodes".alignTable.sequence.status.seqActive;
   "Unit1.Em4.ControlNodes".alignTable."step".action1[180] := #_w1 AND (NOT "Unit1.Em4.ControlNodes".cm.softCam.anodeAlignTableAxisX.waitPos.inPos OR NOT "Unit1.Em4.ControlNodes".cm.softCam.anodeAlignTableAxisY1.waitPos.inPos OR NOT "Unit1.Em4.ControlNodes".cm.softCam.anodeAlignTableAxisY2.waitPos.inPos);
   "Unit1.Em4.ControlNodes".alignTable."step".transition1[180] := #_w1 AND "Unit1.Em4.ControlNodes".cm.softCam.anodeAlignTableAxisX.waitPos.inPos AND "Unit1.Em4.ControlNodes".cm.softCam.anodeAlignTableAxisY1.waitPos.inPos AND "Unit1.Em4.ControlNodes".cm.softCam.anodeAlignTableAxisY2.waitPos.inPos;
   #statTonTime[180].TON(IN := #_w1 AND "Unit1.Em4.ControlNodes".alignTable."step".transition1[180],
                         PT := #delayTime);
   IF #statTonTime[180].Q THEN
       "Unit1.Em4.ControlNodes".alignTable.sequence.status.nextStep := #JOB_1_STEP_90;
   END_IF;
END_REGION

REGION Network 18: Step[181] : Glass Cleaning On
   RUNG wire#powerrail
      { S7_Templates := "SrcType := DInt" } EQ_Contact(in1 := "Unit1.Em4.ControlNodes".alignTable.sequence.status.currentStep, in2 := #JOB_1_STEP_81)
      Contact( "Unit1.Em4.ControlNodes".alignTable.sequence.status.seqActive )
      wire#w1
      Coil( "Unit1.Em4.ControlNodes".alignTable."step".action1[181] )
   END_RUNG
   RUNG wire#w1
      Contact( "Unit1.Em4.HmiInterface".cmAnodeGlassCleaning.monitoring.goToWorkPos )
      wire#w2
      Coil( "Unit1.Em4.ControlNodes".alignTable."step".transition1[181] )
   END_RUNG
   RUNG wire#w1
      Contact( "Unit1.Em4.ControlNodes".alignTable."step".transition1[421] )
   END_RUNG wire#w2
   RUNG wire#w1
      Contact( "Unit1.Em4.ControlNodes".alignTable."step".transition1[181] )
      { S7_Templates := "time_type := Time" } #statTonTime[181].TON(pt := #delayTime, et =>)
      Contact( "Unit1.Em4.ControlNodes".cm.softCam.anodeMainPnP1AxisZ.upPos.inPos )
      Contact( "Unit1.Em4.ControlNodes".cm.softCam.anodeMainPnP2AxisZ.upPos.inPos )
      Move(in := #JOB_1_STEP_90, out1 => "Unit1.Em4.ControlNodes".alignTable.sequence.status.nextStep)
   END_RUNG
   // the same network as SCL:
   "Unit1.Em4.ControlNodes".alignTable."step".action1[181] := ("Unit1.Em4.ControlNodes".alignTable.sequence.status.currentStep = #JOB_1_STEP_81) AND "Unit1.Em4.ControlNodes".alignTable.sequence.status.seqActive;
   "Unit1.Em4.ControlNodes".alignTable."step".transition1[181] := ("Unit1.Em4.ControlNodes".alignTable.sequence.status.currentStep = #JOB_1_STEP_81) AND "Unit1.Em4.ControlNodes".alignTable.sequence.status.seqActive AND ("Unit1.Em4.HmiInterface".cmAnodeGlassCleaning.monitoring.goToWorkPos OR "Unit1.Em4.ControlNodes".alignTable."step".transition1[421]);
   #statTonTime[181].TON(IN := ("Unit1.Em4.ControlNodes".alignTable.sequence.status.currentStep = #JOB_1_STEP_81) AND "Unit1.Em4.ControlNodes".alignTable.sequence.status.seqActive AND "Unit1.Em4.ControlNodes".alignTable."step".transition1[181],
                         PT := #delayTime);
   IF #statTonTime[181].Q AND "Unit1.Em4.ControlNodes".cm.softCam.anodeMainPnP1AxisZ.upPos.inPos AND "Unit1.Em4.ControlNodes".cm.softCam.anodeMainPnP2AxisZ.upPos.inPos THEN
       "Unit1.Em4.ControlNodes".alignTable.sequence.status.nextStep := #JOB_1_STEP_90;
   END_IF;
END_REGION

REGION Network 19: Step[190] : JOB[1] Step End
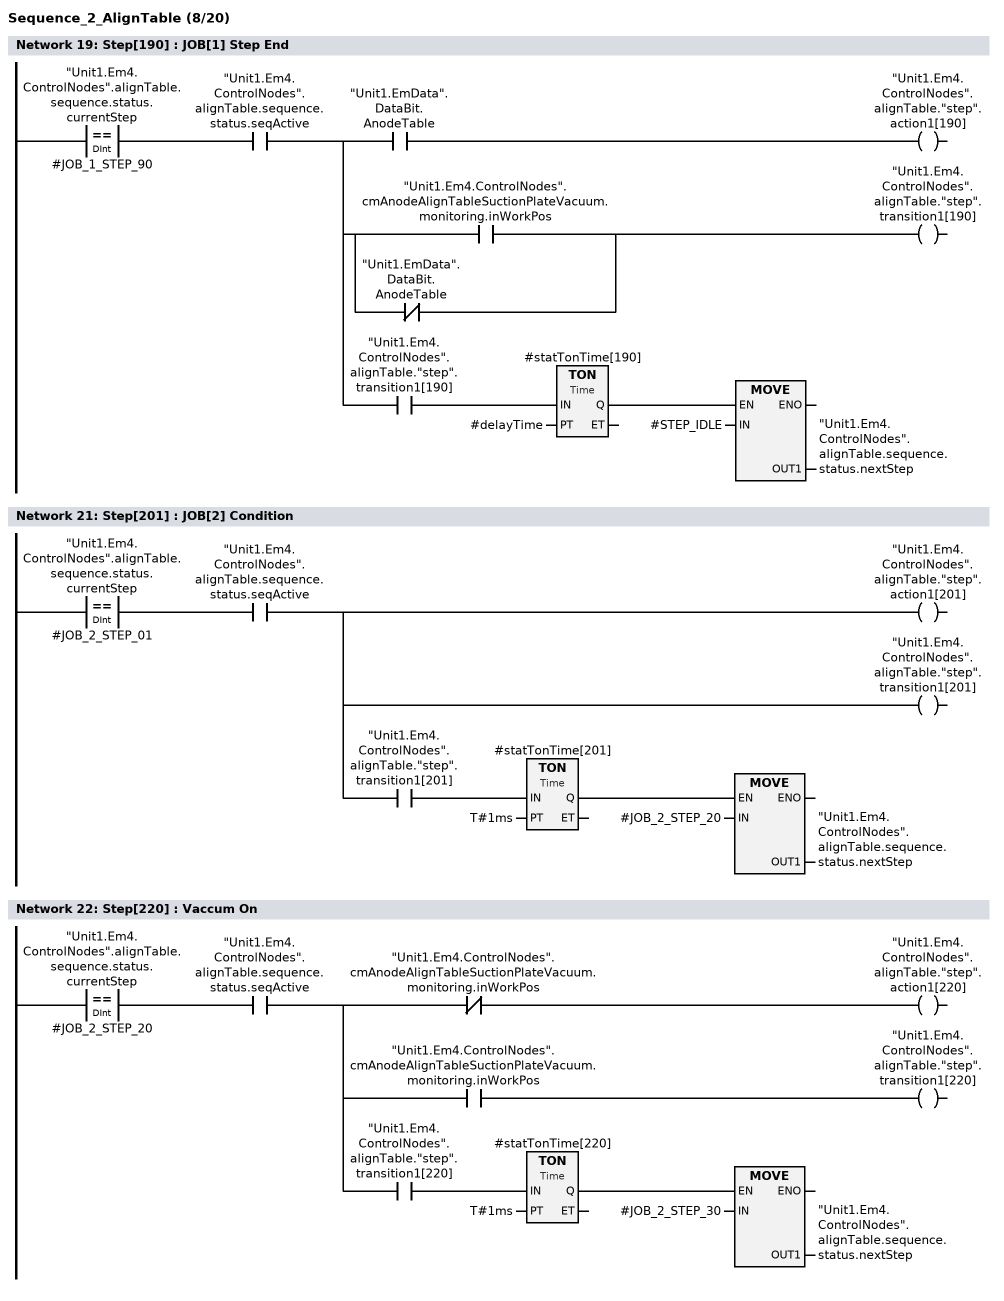
   RUNG wire#powerrail
      { S7_Templates := "SrcType := DInt" } EQ_Contact(in1 := "Unit1.Em4.ControlNodes".alignTable.sequence.status.currentStep, in2 := #JOB_1_STEP_90)
      Contact( "Unit1.Em4.ControlNodes".alignTable.sequence.status.seqActive )
      wire#w1
      Contact( "Unit1.EmData".DataBit.AnodeTable )
      Coil( "Unit1.Em4.ControlNodes".alignTable."step".action1[190] )
   END_RUNG
   RUNG wire#w1
      Contact( "Unit1.Em4.ControlNodes".cmAnodeAlignTableSuctionPlateVacuum.monitoring.inWorkPos )
      wire#w2
      Coil( "Unit1.Em4.ControlNodes".alignTable."step".transition1[190] )
   END_RUNG
   RUNG wire#w1
      I_Contact( "Unit1.EmData".DataBit.AnodeTable )
   END_RUNG wire#w2
   RUNG wire#w1
      Contact( "Unit1.Em4.ControlNodes".alignTable."step".transition1[190] )
      { S7_Templates := "time_type := Time" } #statTonTime[190].TON(pt := #delayTime, et =>)
      Move(in := #STEP_IDLE, out1 => "Unit1.Em4.ControlNodes".alignTable.sequence.status.nextStep)
   END_RUNG
   // the same network as SCL:
   #_w1 := ("Unit1.Em4.ControlNodes".alignTable.sequence.status.currentStep = #JOB_1_STEP_90) AND "Unit1.Em4.ControlNodes".alignTable.sequence.status.seqActive;
   "Unit1.Em4.ControlNodes".alignTable."step".action1[190] := #_w1 AND "Unit1.EmData".DataBit.AnodeTable;
   "Unit1.Em4.ControlNodes".alignTable."step".transition1[190] := #_w1 AND ("Unit1.Em4.ControlNodes".cmAnodeAlignTableSuctionPlateVacuum.monitoring.inWorkPos OR NOT "Unit1.EmData".DataBit.AnodeTable);
   #statTonTime[190].TON(IN := #_w1 AND "Unit1.Em4.ControlNodes".alignTable."step".transition1[190],
                         PT := #delayTime);
   IF #statTonTime[190].Q THEN
       "Unit1.Em4.ControlNodes".alignTable.sequence.status.nextStep := #STEP_IDLE;
   END_IF;
END_REGION

REGION Network 20: ******************** JOB[2] Load ********************
END_REGION

REGION Network 21: Step[201] : JOB[2] Condition
   RUNG wire#powerrail
      { S7_Templates := "SrcType := DInt" } EQ_Contact(in1 := "Unit1.Em4.ControlNodes".alignTable.sequence.status.currentStep, in2 := #JOB_2_STEP_01)
      Contact( "Unit1.Em4.ControlNodes".alignTable.sequence.status.seqActive )
      wire#w1
      Coil( "Unit1.Em4.ControlNodes".alignTable."step".action1[201] )
   END_RUNG
   RUNG wire#w1
      Coil( "Unit1.Em4.ControlNodes".alignTable."step".transition1[201] )
   END_RUNG
   RUNG wire#w1
      Contact( "Unit1.Em4.ControlNodes".alignTable."step".transition1[201] )
      { S7_Templates := "time_type := Time" } #statTonTime[201].TON(pt := T#1ms, et =>)
      Move(in := #JOB_2_STEP_20, out1 => "Unit1.Em4.ControlNodes".alignTable.sequence.status.nextStep)
   END_RUNG
   // the same network as SCL:
   "Unit1.Em4.ControlNodes".alignTable."step".action1[201] := ("Unit1.Em4.ControlNodes".alignTable.sequence.status.currentStep = #JOB_2_STEP_01) AND "Unit1.Em4.ControlNodes".alignTable.sequence.status.seqActive;
   "Unit1.Em4.ControlNodes".alignTable."step".transition1[201] := ("Unit1.Em4.ControlNodes".alignTable.sequence.status.currentStep = #JOB_2_STEP_01) AND "Unit1.Em4.ControlNodes".alignTable.sequence.status.seqActive;
   #statTonTime[201].TON(IN := ("Unit1.Em4.ControlNodes".alignTable.sequence.status.currentStep = #JOB_2_STEP_01) AND "Unit1.Em4.ControlNodes".alignTable.sequence.status.seqActive AND "Unit1.Em4.ControlNodes".alignTable."step".transition1[201],
                         PT := T#1ms);
   IF #statTonTime[201].Q THEN
       "Unit1.Em4.ControlNodes".alignTable.sequence.status.nextStep := #JOB_2_STEP_20;
   END_IF;
END_REGION

REGION Network 22: Step[220] : Vaccum On
   RUNG wire#powerrail
      { S7_Templates := "SrcType := DInt" } EQ_Contact(in1 := "Unit1.Em4.ControlNodes".alignTable.sequence.status.currentStep, in2 := #JOB_2_STEP_20)
      Contact( "Unit1.Em4.ControlNodes".alignTable.sequence.status.seqActive )
      wire#w1
      I_Contact( "Unit1.Em4.ControlNodes".cmAnodeAlignTableSuctionPlateVacuum.monitoring.inWorkPos )
      Coil( "Unit1.Em4.ControlNodes".alignTable."step".action1[220] )
   END_RUNG
   RUNG wire#w1
      Contact( "Unit1.Em4.ControlNodes".cmAnodeAlignTableSuctionPlateVacuum.monitoring.inWorkPos )
      Coil( "Unit1.Em4.ControlNodes".alignTable."step".transition1[220] )
   END_RUNG
   RUNG wire#w1
      Contact( "Unit1.Em4.ControlNodes".alignTable."step".transition1[220] )
      { S7_Templates := "time_type := Time" } #statTonTime[220].TON(pt := T#1ms, et =>)
      Move(in := #JOB_2_STEP_30, out1 => "Unit1.Em4.ControlNodes".alignTable.sequence.status.nextStep)
   END_RUNG
   // the same network as SCL:
   #_w1 := ("Unit1.Em4.ControlNodes".alignTable.sequence.status.currentStep = #JOB_2_STEP_20) AND "Unit1.Em4.ControlNodes".alignTable.sequence.status.seqActive;
   "Unit1.Em4.ControlNodes".alignTable."step".action1[220] := #_w1 AND NOT "Unit1.Em4.ControlNodes".cmAnodeAlignTableSuctionPlateVacuum.monitoring.inWorkPos;
   "Unit1.Em4.ControlNodes".alignTable."step".transition1[220] := #_w1 AND "Unit1.Em4.ControlNodes".cmAnodeAlignTableSuctionPlateVacuum.monitoring.inWorkPos;
   #statTonTime[220].TON(IN := #_w1 AND "Unit1.Em4.ControlNodes".alignTable."step".transition1[220],
                         PT := T#1ms);
   IF #statTonTime[220].Q THEN
       "Unit1.Em4.ControlNodes".alignTable.sequence.status.nextStep := #JOB_2_STEP_30;
   END_IF;
END_REGION

REGION Network 23: Step[230] : Align Table → Main P&P [Load Done]
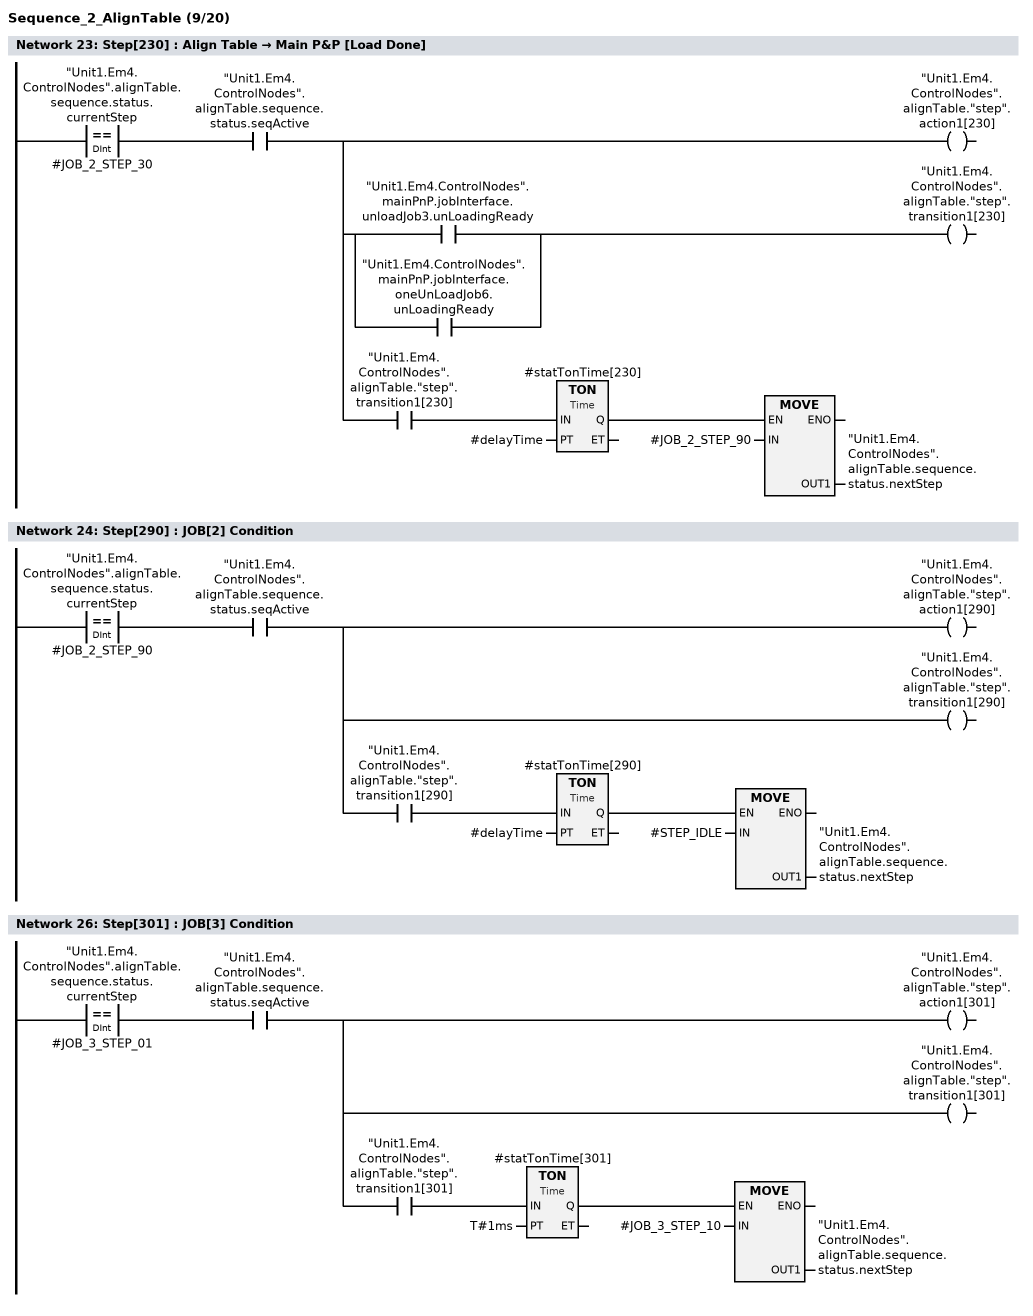
   RUNG wire#powerrail
      { S7_Templates := "SrcType := DInt" } EQ_Contact(in1 := "Unit1.Em4.ControlNodes".alignTable.sequence.status.currentStep, in2 := #JOB_2_STEP_30)
      Contact( "Unit1.Em4.ControlNodes".alignTable.sequence.status.seqActive )
      wire#w1
      Coil( "Unit1.Em4.ControlNodes".alignTable."step".action1[230] )
   END_RUNG
   RUNG wire#w1
      Contact( "Unit1.Em4.ControlNodes".mainPnP.jobInterface.unloadJob3.unLoadingReady )
      wire#w2
      Coil( "Unit1.Em4.ControlNodes".alignTable."step".transition1[230] )
   END_RUNG
   RUNG wire#w1
      Contact( "Unit1.Em4.ControlNodes".mainPnP.jobInterface.oneUnLoadJob6.unLoadingReady )
   END_RUNG wire#w2
   RUNG wire#w1
      Contact( "Unit1.Em4.ControlNodes".alignTable."step".transition1[230] )
      { S7_Templates := "time_type := Time" } #statTonTime[230].TON(pt := #delayTime, et =>)
      Move(in := #JOB_2_STEP_90, out1 => "Unit1.Em4.ControlNodes".alignTable.sequence.status.nextStep)
   END_RUNG
   // the same network as SCL:
   "Unit1.Em4.ControlNodes".alignTable."step".action1[230] := ("Unit1.Em4.ControlNodes".alignTable.sequence.status.currentStep = #JOB_2_STEP_30) AND "Unit1.Em4.ControlNodes".alignTable.sequence.status.seqActive;
   "Unit1.Em4.ControlNodes".alignTable."step".transition1[230] := ("Unit1.Em4.ControlNodes".alignTable.sequence.status.currentStep = #JOB_2_STEP_30) AND "Unit1.Em4.ControlNodes".alignTable.sequence.status.seqActive AND ("Unit1.Em4.ControlNodes".mainPnP.jobInterface.unloadJob3.unLoadingReady OR "Unit1.Em4.ControlNodes".mainPnP.jobInterface.oneUnLoadJob6.unLoadingReady);
   #statTonTime[230].TON(IN := ("Unit1.Em4.ControlNodes".alignTable.sequence.status.currentStep = #JOB_2_STEP_30) AND "Unit1.Em4.ControlNodes".alignTable.sequence.status.seqActive AND "Unit1.Em4.ControlNodes".alignTable."step".transition1[230],
                         PT := #delayTime);
   IF #statTonTime[230].Q THEN
       "Unit1.Em4.ControlNodes".alignTable.sequence.status.nextStep := #JOB_2_STEP_90;
   END_IF;
END_REGION

REGION Network 24: Step[290] : JOB[2] Condition
   RUNG wire#powerrail
      { S7_Templates := "SrcType := DInt" } EQ_Contact(in1 := "Unit1.Em4.ControlNodes".alignTable.sequence.status.currentStep, in2 := #JOB_2_STEP_90)
      Contact( "Unit1.Em4.ControlNodes".alignTable.sequence.status.seqActive )
      wire#w1
      Coil( "Unit1.Em4.ControlNodes".alignTable."step".action1[290] )
   END_RUNG
   RUNG wire#w1
      Coil( "Unit1.Em4.ControlNodes".alignTable."step".transition1[290] )
   END_RUNG
   RUNG wire#w1
      Contact( "Unit1.Em4.ControlNodes".alignTable."step".transition1[290] )
      { S7_Templates := "time_type := Time" } #statTonTime[290].TON(pt := #delayTime, et =>)
      Move(in := #STEP_IDLE, out1 => "Unit1.Em4.ControlNodes".alignTable.sequence.status.nextStep)
   END_RUNG
   // the same network as SCL:
   "Unit1.Em4.ControlNodes".alignTable."step".action1[290] := ("Unit1.Em4.ControlNodes".alignTable.sequence.status.currentStep = #JOB_2_STEP_90) AND "Unit1.Em4.ControlNodes".alignTable.sequence.status.seqActive;
   "Unit1.Em4.ControlNodes".alignTable."step".transition1[290] := ("Unit1.Em4.ControlNodes".alignTable.sequence.status.currentStep = #JOB_2_STEP_90) AND "Unit1.Em4.ControlNodes".alignTable.sequence.status.seqActive;
   #statTonTime[290].TON(IN := ("Unit1.Em4.ControlNodes".alignTable.sequence.status.currentStep = #JOB_2_STEP_90) AND "Unit1.Em4.ControlNodes".alignTable.sequence.status.seqActive AND "Unit1.Em4.ControlNodes".alignTable."step".transition1[290],
                         PT := #delayTime);
   IF #statTonTime[290].Q THEN
       "Unit1.Em4.ControlNodes".alignTable.sequence.status.nextStep := #STEP_IDLE;
   END_IF;
END_REGION

REGION Network 25: ******************** JOB[3] Vision ********************
END_REGION

REGION Network 26: Step[301] : JOB[3] Condition
   RUNG wire#powerrail
      { S7_Templates := "SrcType := DInt" } EQ_Contact(in1 := "Unit1.Em4.ControlNodes".alignTable.sequence.status.currentStep, in2 := #JOB_3_STEP_01)
      Contact( "Unit1.Em4.ControlNodes".alignTable.sequence.status.seqActive )
      wire#w1
      Coil( "Unit1.Em4.ControlNodes".alignTable."step".action1[301] )
   END_RUNG
   RUNG wire#w1
      Coil( "Unit1.Em4.ControlNodes".alignTable."step".transition1[301] )
   END_RUNG
   RUNG wire#w1
      Contact( "Unit1.Em4.ControlNodes".alignTable."step".transition1[301] )
      { S7_Templates := "time_type := Time" } #statTonTime[301].TON(pt := T#1ms, et =>)
      Move(in := #JOB_3_STEP_10, out1 => "Unit1.Em4.ControlNodes".alignTable.sequence.status.nextStep)
   END_RUNG
   // the same network as SCL:
   "Unit1.Em4.ControlNodes".alignTable."step".action1[301] := ("Unit1.Em4.ControlNodes".alignTable.sequence.status.currentStep = #JOB_3_STEP_01) AND "Unit1.Em4.ControlNodes".alignTable.sequence.status.seqActive;
   "Unit1.Em4.ControlNodes".alignTable."step".transition1[301] := ("Unit1.Em4.ControlNodes".alignTable.sequence.status.currentStep = #JOB_3_STEP_01) AND "Unit1.Em4.ControlNodes".alignTable.sequence.status.seqActive;
   #statTonTime[301].TON(IN := ("Unit1.Em4.ControlNodes".alignTable.sequence.status.currentStep = #JOB_3_STEP_01) AND "Unit1.Em4.ControlNodes".alignTable.sequence.status.seqActive AND "Unit1.Em4.ControlNodes".alignTable."step".transition1[301],
                         PT := T#1ms);
   IF #statTonTime[301].Q THEN
       "Unit1.Em4.ControlNodes".alignTable.sequence.status.nextStep := #JOB_3_STEP_10;
   END_IF;
END_REGION

REGION Network 27: Step[310] : Vision Start
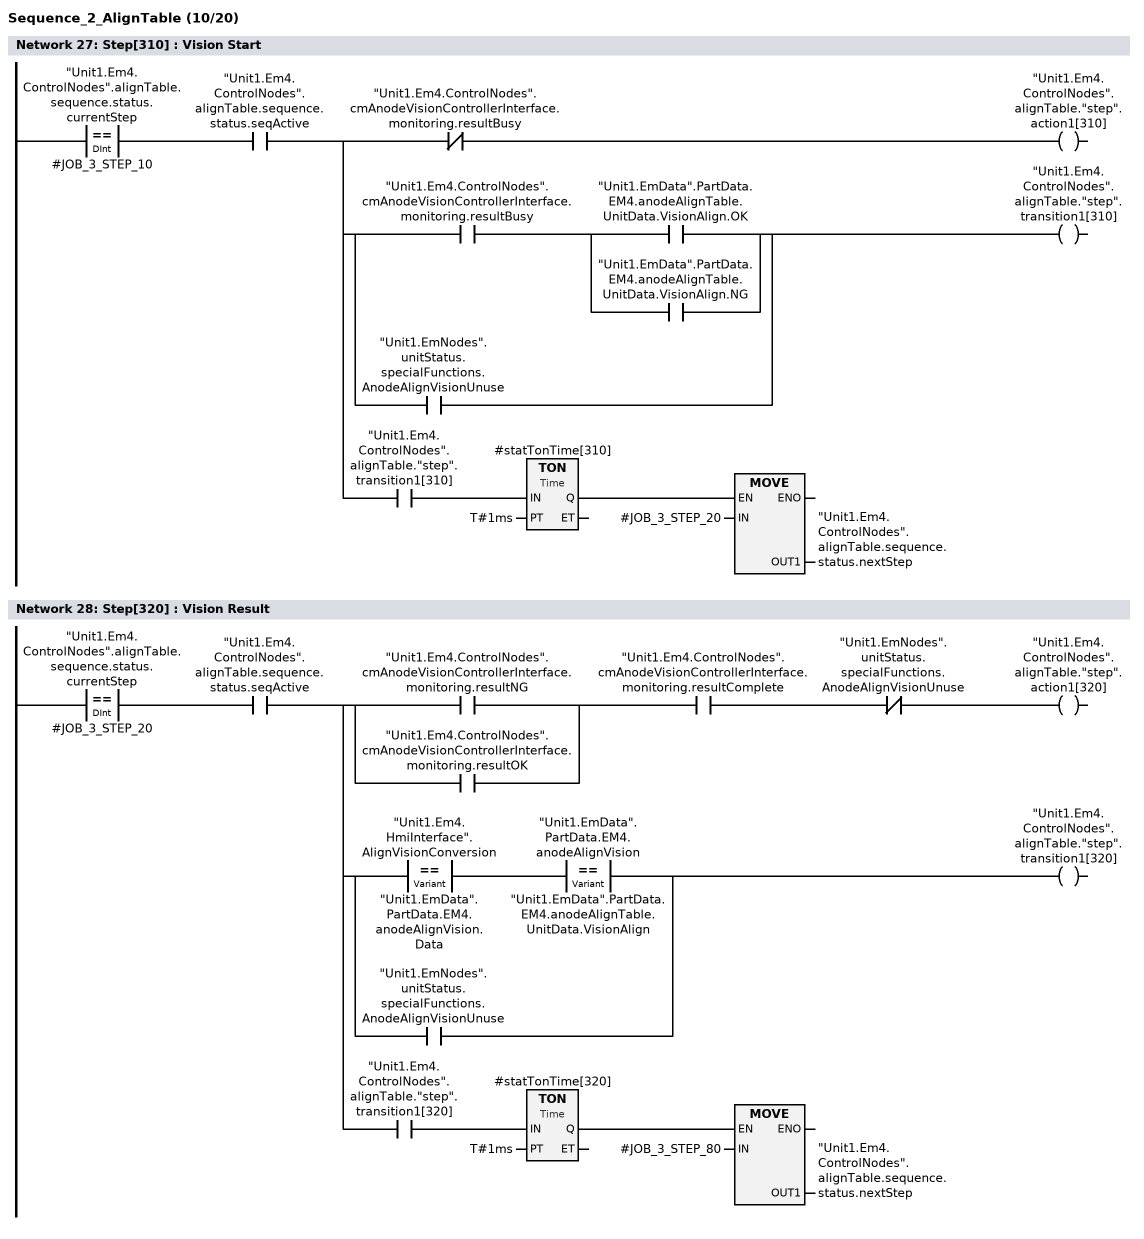
   RUNG wire#powerrail
      { S7_Templates := "SrcType := DInt" } EQ_Contact(in1 := "Unit1.Em4.ControlNodes".alignTable.sequence.status.currentStep, in2 := #JOB_3_STEP_10)
      Contact( "Unit1.Em4.ControlNodes".alignTable.sequence.status.seqActive )
      wire#w1
      I_Contact( "Unit1.Em4.ControlNodes".cmAnodeVisionControllerInterface.monitoring.resultBusy )
      Coil( "Unit1.Em4.ControlNodes".alignTable."step".action1[310] )
   END_RUNG
   RUNG wire#w1
      Contact( "Unit1.Em4.ControlNodes".cmAnodeVisionControllerInterface.monitoring.resultBusy )
      wire#w2
      Contact( "Unit1.EmData".PartData.EM4.anodeAlignTable.UnitData.VisionAlign.OK )
      wire#w3
      Coil( "Unit1.Em4.ControlNodes".alignTable."step".transition1[310] )
   END_RUNG
   RUNG wire#w2
      Contact( "Unit1.EmData".PartData.EM4.anodeAlignTable.UnitData.VisionAlign.NG )
   END_RUNG wire#w3
   RUNG wire#w1
      Contact( "Unit1.EmNodes".unitStatus.specialFunctions.AnodeAlignVisionUnuse )
   END_RUNG wire#w3
   RUNG wire#w1
      Contact( "Unit1.Em4.ControlNodes".alignTable."step".transition1[310] )
      { S7_Templates := "time_type := Time" } #statTonTime[310].TON(pt := T#1ms, et =>)
      Move(in := #JOB_3_STEP_20, out1 => "Unit1.Em4.ControlNodes".alignTable.sequence.status.nextStep)
   END_RUNG
   // the same network as SCL:
   #_w1 := ("Unit1.Em4.ControlNodes".alignTable.sequence.status.currentStep = #JOB_3_STEP_10) AND "Unit1.Em4.ControlNodes".alignTable.sequence.status.seqActive;
   "Unit1.Em4.ControlNodes".alignTable."step".action1[310] := #_w1 AND NOT "Unit1.Em4.ControlNodes".cmAnodeVisionControllerInterface.monitoring.resultBusy;
   "Unit1.Em4.ControlNodes".alignTable."step".transition1[310] := #_w1 AND (("Unit1.Em4.ControlNodes".cmAnodeVisionControllerInterface.monitoring.resultBusy AND ("Unit1.EmData".PartData.EM4.anodeAlignTable.UnitData.VisionAlign.OK OR "Unit1.EmData".PartData.EM4.anodeAlignTable.UnitData.VisionAlign.NG)) OR "Unit1.EmNodes".unitStatus.specialFunctions.AnodeAlignVisionUnuse);
   #statTonTime[310].TON(IN := #_w1 AND "Unit1.Em4.ControlNodes".alignTable."step".transition1[310],
                         PT := T#1ms);
   IF #statTonTime[310].Q THEN
       "Unit1.Em4.ControlNodes".alignTable.sequence.status.nextStep := #JOB_3_STEP_20;
   END_IF;
END_REGION

REGION Network 28: Step[320] : Vision Result
   RUNG wire#powerrail
      { S7_Templates := "SrcType := DInt" } EQ_Contact(in1 := "Unit1.Em4.ControlNodes".alignTable.sequence.status.currentStep, in2 := #JOB_3_STEP_20)
      Contact( "Unit1.Em4.ControlNodes".alignTable.sequence.status.seqActive )
      wire#w1
      Contact( "Unit1.Em4.ControlNodes".cmAnodeVisionControllerInterface.monitoring.resultNG )
      wire#w2
      Contact( "Unit1.Em4.ControlNodes".cmAnodeVisionControllerInterface.monitoring.resultComplete )
      I_Contact( "Unit1.EmNodes".unitStatus.specialFunctions.AnodeAlignVisionUnuse )
      Coil( "Unit1.Em4.ControlNodes".alignTable."step".action1[320] )
   END_RUNG
   RUNG wire#w1
      Contact( "Unit1.Em4.ControlNodes".cmAnodeVisionControllerInterface.monitoring.resultOK )
   END_RUNG wire#w2
   RUNG wire#w1
      { S7_Templates := "SrcType := Variant" } EQ_Contact(in1 := "Unit1.Em4.HmiInterface".AlignVisionConversion, in2 := "Unit1.EmData".PartData.EM4.anodeAlignVision.Data)
      { S7_Templates := "SrcType := Variant" } EQ_Contact(in1 := "Unit1.EmData".PartData.EM4.anodeAlignVision, in2 := "Unit1.EmData".PartData.EM4.anodeAlignTable.UnitData.VisionAlign)
      wire#w3
      Coil( "Unit1.Em4.ControlNodes".alignTable."step".transition1[320] )
   END_RUNG
   RUNG wire#w1
      Contact( "Unit1.EmNodes".unitStatus.specialFunctions.AnodeAlignVisionUnuse )
   END_RUNG wire#w3
   RUNG wire#w1
      Contact( "Unit1.Em4.ControlNodes".alignTable."step".transition1[320] )
      { S7_Templates := "time_type := Time" } #statTonTime[320].TON(pt := T#1ms, et =>)
      Move(in := #JOB_3_STEP_80, out1 => "Unit1.Em4.ControlNodes".alignTable.sequence.status.nextStep)
   END_RUNG
   // the same network as SCL:
   #_w1 := ("Unit1.Em4.ControlNodes".alignTable.sequence.status.currentStep = #JOB_3_STEP_20) AND "Unit1.Em4.ControlNodes".alignTable.sequence.status.seqActive;
   "Unit1.Em4.ControlNodes".alignTable."step".action1[320] := #_w1 AND ("Unit1.Em4.ControlNodes".cmAnodeVisionControllerInterface.monitoring.resultNG OR "Unit1.Em4.ControlNodes".cmAnodeVisionControllerInterface.monitoring.resultOK) AND "Unit1.Em4.ControlNodes".cmAnodeVisionControllerInterface.monitoring.resultComplete AND NOT "Unit1.EmNodes".unitStatus.specialFunctions.AnodeAlignVisionUnuse;
   "Unit1.Em4.ControlNodes".alignTable."step".transition1[320] := #_w1 AND ((("Unit1.Em4.HmiInterface".AlignVisionConversion = "Unit1.EmData".PartData.EM4.anodeAlignVision.Data) AND ("Unit1.EmData".PartData.EM4.anodeAlignVision = "Unit1.EmData".PartData.EM4.anodeAlignTable.UnitData.VisionAlign)) OR "Unit1.EmNodes".unitStatus.specialFunctions.AnodeAlignVisionUnuse);
   #statTonTime[320].TON(IN := #_w1 AND "Unit1.Em4.ControlNodes".alignTable."step".transition1[320],
                         PT := T#1ms);
   IF #statTonTime[320].Q THEN
       "Unit1.Em4.ControlNodes".alignTable.sequence.status.nextStep := #JOB_3_STEP_80;
   END_IF;
END_REGION

REGION Network 29: Step[380] : Align Table X,Y1,Y2-Axis Work Pos
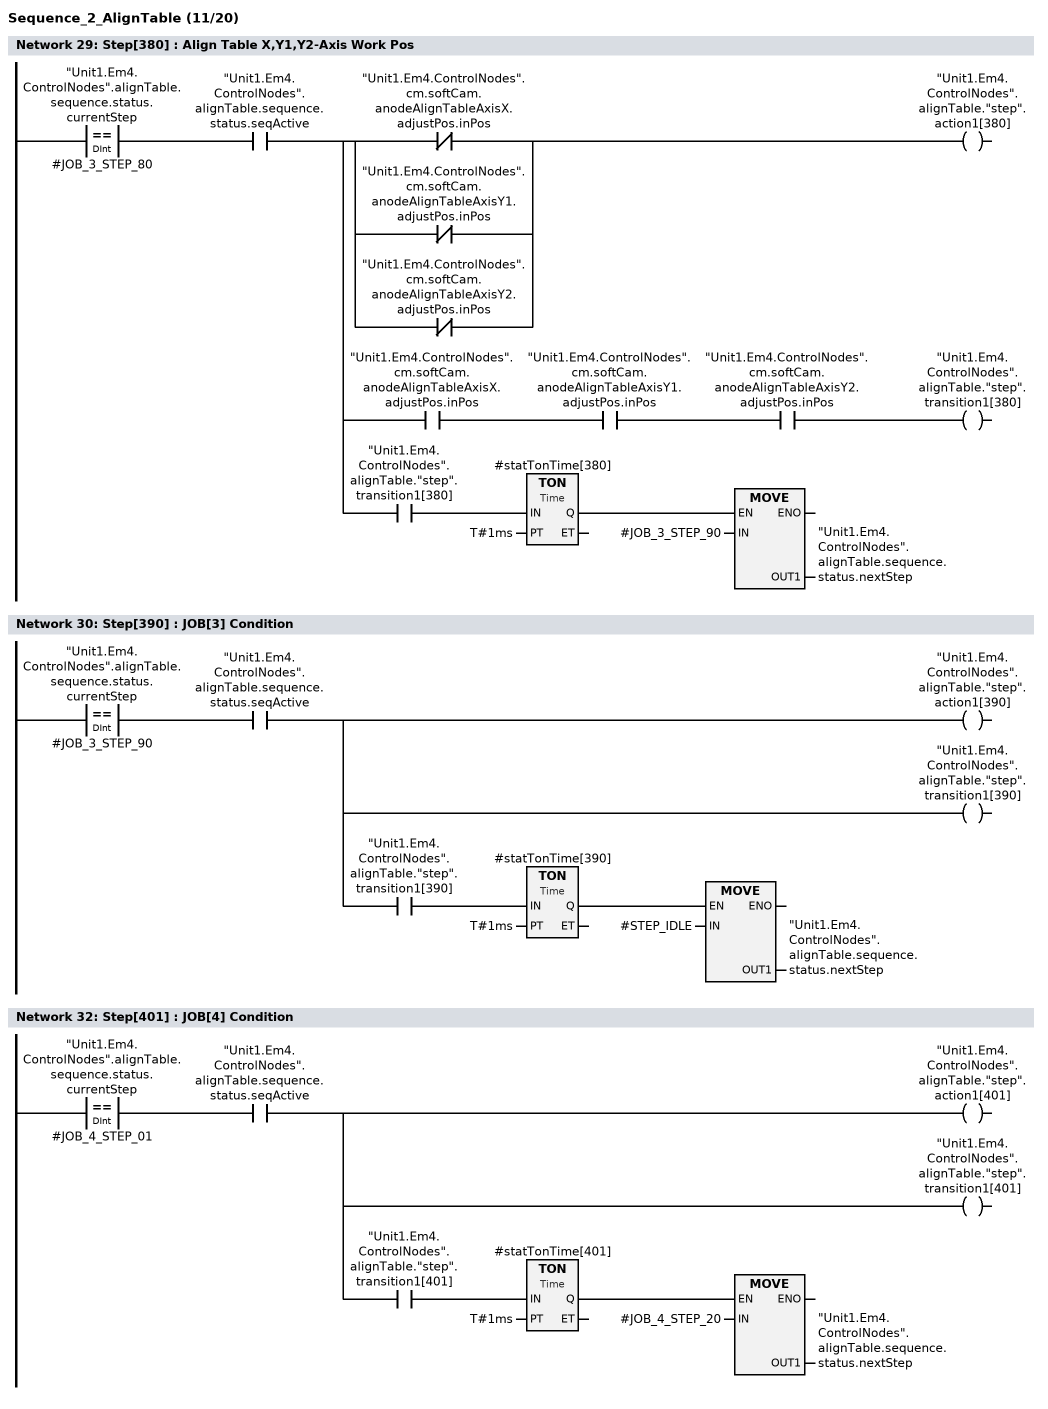
   RUNG wire#powerrail
      { S7_Templates := "SrcType := DInt" } EQ_Contact(in1 := "Unit1.Em4.ControlNodes".alignTable.sequence.status.currentStep, in2 := #JOB_3_STEP_80)
      Contact( "Unit1.Em4.ControlNodes".alignTable.sequence.status.seqActive )
      wire#w1
      I_Contact( "Unit1.Em4.ControlNodes".cm.softCam.anodeAlignTableAxisX.adjustPos.inPos )
      wire#w2
      Coil( "Unit1.Em4.ControlNodes".alignTable."step".action1[380] )
   END_RUNG
   RUNG wire#w1
      I_Contact( "Unit1.Em4.ControlNodes".cm.softCam.anodeAlignTableAxisY1.adjustPos.inPos )
   END_RUNG wire#w2
   RUNG wire#w1
      I_Contact( "Unit1.Em4.ControlNodes".cm.softCam.anodeAlignTableAxisY2.adjustPos.inPos )
   END_RUNG wire#w2
   RUNG wire#w1
      Contact( "Unit1.Em4.ControlNodes".cm.softCam.anodeAlignTableAxisX.adjustPos.inPos )
      Contact( "Unit1.Em4.ControlNodes".cm.softCam.anodeAlignTableAxisY1.adjustPos.inPos )
      Contact( "Unit1.Em4.ControlNodes".cm.softCam.anodeAlignTableAxisY2.adjustPos.inPos )
      Coil( "Unit1.Em4.ControlNodes".alignTable."step".transition1[380] )
   END_RUNG
   RUNG wire#w1
      Contact( "Unit1.Em4.ControlNodes".alignTable."step".transition1[380] )
      { S7_Templates := "time_type := Time" } #statTonTime[380].TON(pt := T#1ms, et =>)
      Move(in := #JOB_3_STEP_90, out1 => "Unit1.Em4.ControlNodes".alignTable.sequence.status.nextStep)
   END_RUNG
   // the same network as SCL:
   #_w1 := ("Unit1.Em4.ControlNodes".alignTable.sequence.status.currentStep = #JOB_3_STEP_80) AND "Unit1.Em4.ControlNodes".alignTable.sequence.status.seqActive;
   "Unit1.Em4.ControlNodes".alignTable."step".action1[380] := #_w1 AND (NOT "Unit1.Em4.ControlNodes".cm.softCam.anodeAlignTableAxisX.adjustPos.inPos OR NOT "Unit1.Em4.ControlNodes".cm.softCam.anodeAlignTableAxisY1.adjustPos.inPos OR NOT "Unit1.Em4.ControlNodes".cm.softCam.anodeAlignTableAxisY2.adjustPos.inPos);
   "Unit1.Em4.ControlNodes".alignTable."step".transition1[380] := #_w1 AND "Unit1.Em4.ControlNodes".cm.softCam.anodeAlignTableAxisX.adjustPos.inPos AND "Unit1.Em4.ControlNodes".cm.softCam.anodeAlignTableAxisY1.adjustPos.inPos AND "Unit1.Em4.ControlNodes".cm.softCam.anodeAlignTableAxisY2.adjustPos.inPos;
   #statTonTime[380].TON(IN := #_w1 AND "Unit1.Em4.ControlNodes".alignTable."step".transition1[380],
                         PT := T#1ms);
   IF #statTonTime[380].Q THEN
       "Unit1.Em4.ControlNodes".alignTable.sequence.status.nextStep := #JOB_3_STEP_90;
   END_IF;
END_REGION

REGION Network 30: Step[390] : JOB[3] Condition
   RUNG wire#powerrail
      { S7_Templates := "SrcType := DInt" } EQ_Contact(in1 := "Unit1.Em4.ControlNodes".alignTable.sequence.status.currentStep, in2 := #JOB_3_STEP_90)
      Contact( "Unit1.Em4.ControlNodes".alignTable.sequence.status.seqActive )
      wire#w1
      Coil( "Unit1.Em4.ControlNodes".alignTable."step".action1[390] )
   END_RUNG
   RUNG wire#w1
      Coil( "Unit1.Em4.ControlNodes".alignTable."step".transition1[390] )
   END_RUNG
   RUNG wire#w1
      Contact( "Unit1.Em4.ControlNodes".alignTable."step".transition1[390] )
      { S7_Templates := "time_type := Time" } #statTonTime[390].TON(pt := T#1ms, et =>)
      Move(in := #STEP_IDLE, out1 => "Unit1.Em4.ControlNodes".alignTable.sequence.status.nextStep)
   END_RUNG
   // the same network as SCL:
   "Unit1.Em4.ControlNodes".alignTable."step".action1[390] := ("Unit1.Em4.ControlNodes".alignTable.sequence.status.currentStep = #JOB_3_STEP_90) AND "Unit1.Em4.ControlNodes".alignTable.sequence.status.seqActive;
   "Unit1.Em4.ControlNodes".alignTable."step".transition1[390] := ("Unit1.Em4.ControlNodes".alignTable.sequence.status.currentStep = #JOB_3_STEP_90) AND "Unit1.Em4.ControlNodes".alignTable.sequence.status.seqActive;
   #statTonTime[390].TON(IN := ("Unit1.Em4.ControlNodes".alignTable.sequence.status.currentStep = #JOB_3_STEP_90) AND "Unit1.Em4.ControlNodes".alignTable.sequence.status.seqActive AND "Unit1.Em4.ControlNodes".alignTable."step".transition1[390],
                         PT := T#1ms);
   IF #statTonTime[390].Q THEN
       "Unit1.Em4.ControlNodes".alignTable.sequence.status.nextStep := #STEP_IDLE;
   END_IF;
END_REGION

REGION Network 31: ******************** JOB[4] Unload ********************
END_REGION

REGION Network 32: Step[401] : JOB[4] Condition
   RUNG wire#powerrail
      { S7_Templates := "SrcType := DInt" } EQ_Contact(in1 := "Unit1.Em4.ControlNodes".alignTable.sequence.status.currentStep, in2 := #JOB_4_STEP_01)
      Contact( "Unit1.Em4.ControlNodes".alignTable.sequence.status.seqActive )
      wire#w1
      Coil( "Unit1.Em4.ControlNodes".alignTable."step".action1[401] )
   END_RUNG
   RUNG wire#w1
      Coil( "Unit1.Em4.ControlNodes".alignTable."step".transition1[401] )
   END_RUNG
   RUNG wire#w1
      Contact( "Unit1.Em4.ControlNodes".alignTable."step".transition1[401] )
      { S7_Templates := "time_type := Time" } #statTonTime[401].TON(pt := T#1ms, et =>)
      Move(in := #JOB_4_STEP_20, out1 => "Unit1.Em4.ControlNodes".alignTable.sequence.status.nextStep)
   END_RUNG
   // the same network as SCL:
   "Unit1.Em4.ControlNodes".alignTable."step".action1[401] := ("Unit1.Em4.ControlNodes".alignTable.sequence.status.currentStep = #JOB_4_STEP_01) AND "Unit1.Em4.ControlNodes".alignTable.sequence.status.seqActive;
   "Unit1.Em4.ControlNodes".alignTable."step".transition1[401] := ("Unit1.Em4.ControlNodes".alignTable.sequence.status.currentStep = #JOB_4_STEP_01) AND "Unit1.Em4.ControlNodes".alignTable.sequence.status.seqActive;
   #statTonTime[401].TON(IN := ("Unit1.Em4.ControlNodes".alignTable.sequence.status.currentStep = #JOB_4_STEP_01) AND "Unit1.Em4.ControlNodes".alignTable.sequence.status.seqActive AND "Unit1.Em4.ControlNodes".alignTable."step".transition1[401],
                         PT := T#1ms);
   IF #statTonTime[401].Q THEN
       "Unit1.Em4.ControlNodes".alignTable.sequence.status.nextStep := #JOB_4_STEP_20;
   END_IF;
END_REGION

REGION Network 33: Step[420] : Vaccum Off
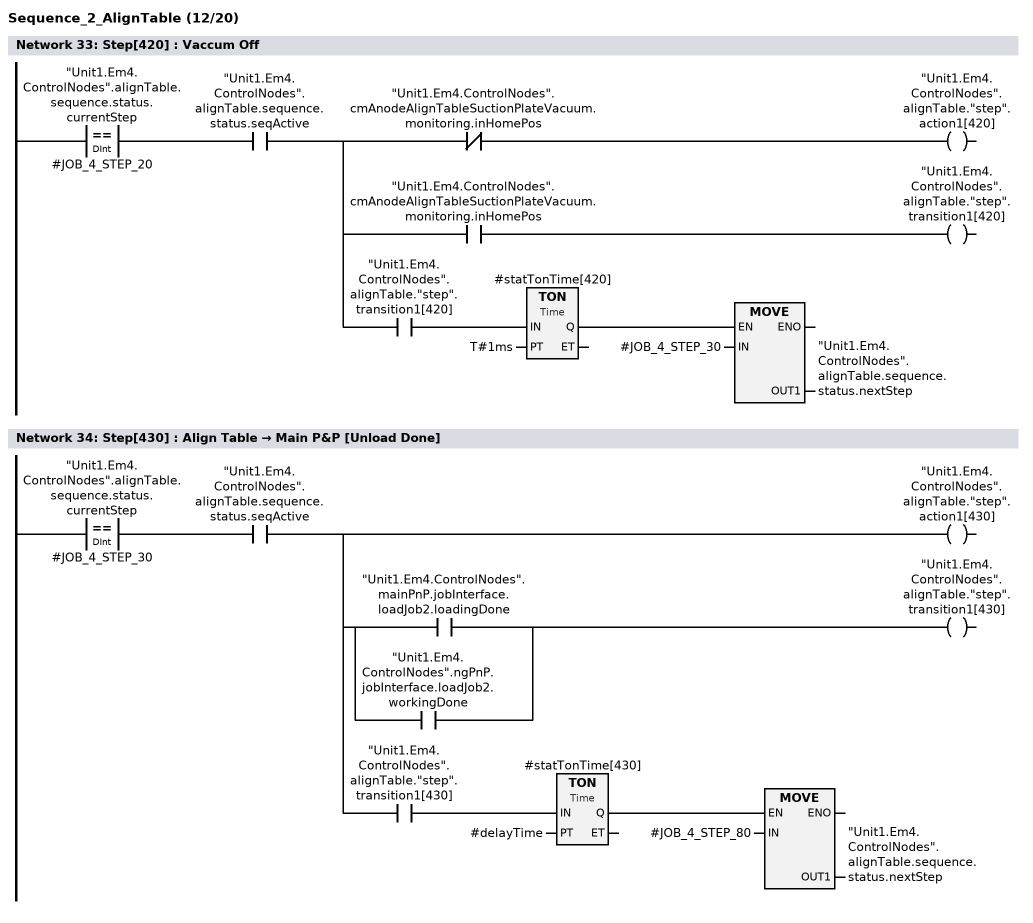
   RUNG wire#powerrail
      { S7_Templates := "SrcType := DInt" } EQ_Contact(in1 := "Unit1.Em4.ControlNodes".alignTable.sequence.status.currentStep, in2 := #JOB_4_STEP_20)
      Contact( "Unit1.Em4.ControlNodes".alignTable.sequence.status.seqActive )
      wire#w1
      I_Contact( "Unit1.Em4.ControlNodes".cmAnodeAlignTableSuctionPlateVacuum.monitoring.inHomePos )
      Coil( "Unit1.Em4.ControlNodes".alignTable."step".action1[420] )
   END_RUNG
   RUNG wire#w1
      Contact( "Unit1.Em4.ControlNodes".cmAnodeAlignTableSuctionPlateVacuum.monitoring.inHomePos )
      Coil( "Unit1.Em4.ControlNodes".alignTable."step".transition1[420] )
   END_RUNG
   RUNG wire#w1
      Contact( "Unit1.Em4.ControlNodes".alignTable."step".transition1[420] )
      { S7_Templates := "time_type := Time" } #statTonTime[420].TON(pt := T#1ms, et =>)
      Move(in := #JOB_4_STEP_30, out1 => "Unit1.Em4.ControlNodes".alignTable.sequence.status.nextStep)
   END_RUNG
   // the same network as SCL:
   #_w1 := ("Unit1.Em4.ControlNodes".alignTable.sequence.status.currentStep = #JOB_4_STEP_20) AND "Unit1.Em4.ControlNodes".alignTable.sequence.status.seqActive;
   "Unit1.Em4.ControlNodes".alignTable."step".action1[420] := #_w1 AND NOT "Unit1.Em4.ControlNodes".cmAnodeAlignTableSuctionPlateVacuum.monitoring.inHomePos;
   "Unit1.Em4.ControlNodes".alignTable."step".transition1[420] := #_w1 AND "Unit1.Em4.ControlNodes".cmAnodeAlignTableSuctionPlateVacuum.monitoring.inHomePos;
   #statTonTime[420].TON(IN := #_w1 AND "Unit1.Em4.ControlNodes".alignTable."step".transition1[420],
                         PT := T#1ms);
   IF #statTonTime[420].Q THEN
       "Unit1.Em4.ControlNodes".alignTable.sequence.status.nextStep := #JOB_4_STEP_30;
   END_IF;
END_REGION

REGION Network 34: Step[430] : Align Table → Main P&P [Unload Done]
   RUNG wire#powerrail
      { S7_Templates := "SrcType := DInt" } EQ_Contact(in1 := "Unit1.Em4.ControlNodes".alignTable.sequence.status.currentStep, in2 := #JOB_4_STEP_30)
      Contact( "Unit1.Em4.ControlNodes".alignTable.sequence.status.seqActive )
      wire#w1
      Coil( "Unit1.Em4.ControlNodes".alignTable."step".action1[430] )
   END_RUNG
   RUNG wire#w1
      Contact( "Unit1.Em4.ControlNodes".mainPnP.jobInterface.loadJob2.loadingDone )
      wire#w2
      Coil( "Unit1.Em4.ControlNodes".alignTable."step".transition1[430] )
   END_RUNG
   RUNG wire#w1
      Contact( "Unit1.Em4.ControlNodes".ngPnP.jobInterface.loadJob2.workingDone )
   END_RUNG wire#w2
   RUNG wire#w1
      Contact( "Unit1.Em4.ControlNodes".alignTable."step".transition1[430] )
      { S7_Templates := "time_type := Time" } #statTonTime[430].TON(pt := #delayTime, et =>)
      Move(in := #JOB_4_STEP_80, out1 => "Unit1.Em4.ControlNodes".alignTable.sequence.status.nextStep)
   END_RUNG
   // the same network as SCL:
   "Unit1.Em4.ControlNodes".alignTable."step".action1[430] := ("Unit1.Em4.ControlNodes".alignTable.sequence.status.currentStep = #JOB_4_STEP_30) AND "Unit1.Em4.ControlNodes".alignTable.sequence.status.seqActive;
   "Unit1.Em4.ControlNodes".alignTable."step".transition1[430] := ("Unit1.Em4.ControlNodes".alignTable.sequence.status.currentStep = #JOB_4_STEP_30) AND "Unit1.Em4.ControlNodes".alignTable.sequence.status.seqActive AND ("Unit1.Em4.ControlNodes".mainPnP.jobInterface.loadJob2.loadingDone OR "Unit1.Em4.ControlNodes".ngPnP.jobInterface.loadJob2.workingDone);
   #statTonTime[430].TON(IN := ("Unit1.Em4.ControlNodes".alignTable.sequence.status.currentStep = #JOB_4_STEP_30) AND "Unit1.Em4.ControlNodes".alignTable.sequence.status.seqActive AND "Unit1.Em4.ControlNodes".alignTable."step".transition1[430],
                         PT := #delayTime);
   IF #statTonTime[430].Q THEN
       "Unit1.Em4.ControlNodes".alignTable.sequence.status.nextStep := #JOB_4_STEP_80;
   END_IF;
END_REGION

REGION Network 35: Step[480] : Align Table X,Y1,Y2-Axis Wait Pos
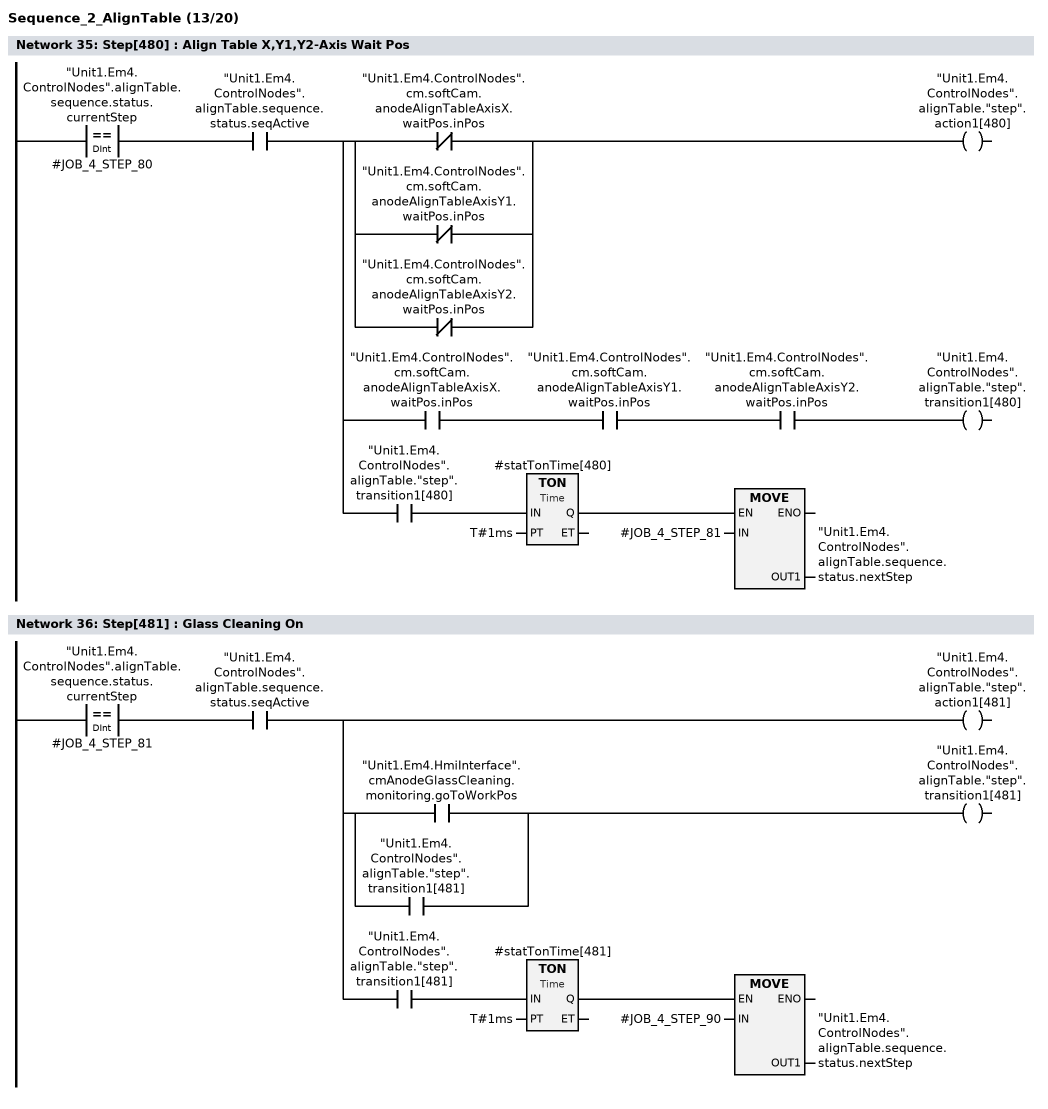
   RUNG wire#powerrail
      { S7_Templates := "SrcType := DInt" } EQ_Contact(in1 := "Unit1.Em4.ControlNodes".alignTable.sequence.status.currentStep, in2 := #JOB_4_STEP_80)
      Contact( "Unit1.Em4.ControlNodes".alignTable.sequence.status.seqActive )
      wire#w1
      I_Contact( "Unit1.Em4.ControlNodes".cm.softCam.anodeAlignTableAxisX.waitPos.inPos )
      wire#w2
      Coil( "Unit1.Em4.ControlNodes".alignTable."step".action1[480] )
   END_RUNG
   RUNG wire#w1
      I_Contact( "Unit1.Em4.ControlNodes".cm.softCam.anodeAlignTableAxisY1.waitPos.inPos )
   END_RUNG wire#w2
   RUNG wire#w1
      I_Contact( "Unit1.Em4.ControlNodes".cm.softCam.anodeAlignTableAxisY2.waitPos.inPos )
   END_RUNG wire#w2
   RUNG wire#w1
      Contact( "Unit1.Em4.ControlNodes".cm.softCam.anodeAlignTableAxisX.waitPos.inPos )
      Contact( "Unit1.Em4.ControlNodes".cm.softCam.anodeAlignTableAxisY1.waitPos.inPos )
      Contact( "Unit1.Em4.ControlNodes".cm.softCam.anodeAlignTableAxisY2.waitPos.inPos )
      Coil( "Unit1.Em4.ControlNodes".alignTable."step".transition1[480] )
   END_RUNG
   RUNG wire#w1
      Contact( "Unit1.Em4.ControlNodes".alignTable."step".transition1[480] )
      { S7_Templates := "time_type := Time" } #statTonTime[480].TON(pt := T#1ms, et =>)
      Move(in := #JOB_4_STEP_81, out1 => "Unit1.Em4.ControlNodes".alignTable.sequence.status.nextStep)
   END_RUNG
   // the same network as SCL:
   #_w1 := ("Unit1.Em4.ControlNodes".alignTable.sequence.status.currentStep = #JOB_4_STEP_80) AND "Unit1.Em4.ControlNodes".alignTable.sequence.status.seqActive;
   "Unit1.Em4.ControlNodes".alignTable."step".action1[480] := #_w1 AND (NOT "Unit1.Em4.ControlNodes".cm.softCam.anodeAlignTableAxisX.waitPos.inPos OR NOT "Unit1.Em4.ControlNodes".cm.softCam.anodeAlignTableAxisY1.waitPos.inPos OR NOT "Unit1.Em4.ControlNodes".cm.softCam.anodeAlignTableAxisY2.waitPos.inPos);
   "Unit1.Em4.ControlNodes".alignTable."step".transition1[480] := #_w1 AND "Unit1.Em4.ControlNodes".cm.softCam.anodeAlignTableAxisX.waitPos.inPos AND "Unit1.Em4.ControlNodes".cm.softCam.anodeAlignTableAxisY1.waitPos.inPos AND "Unit1.Em4.ControlNodes".cm.softCam.anodeAlignTableAxisY2.waitPos.inPos;
   #statTonTime[480].TON(IN := #_w1 AND "Unit1.Em4.ControlNodes".alignTable."step".transition1[480],
                         PT := T#1ms);
   IF #statTonTime[480].Q THEN
       "Unit1.Em4.ControlNodes".alignTable.sequence.status.nextStep := #JOB_4_STEP_81;
   END_IF;
END_REGION

REGION Network 36: Step[481] : Glass Cleaning On
   RUNG wire#powerrail
      { S7_Templates := "SrcType := DInt" } EQ_Contact(in1 := "Unit1.Em4.ControlNodes".alignTable.sequence.status.currentStep, in2 := #JOB_4_STEP_81)
      Contact( "Unit1.Em4.ControlNodes".alignTable.sequence.status.seqActive )
      wire#w1
      Coil( "Unit1.Em4.ControlNodes".alignTable."step".action1[481] )
   END_RUNG
   RUNG wire#w1
      Contact( "Unit1.Em4.HmiInterface".cmAnodeGlassCleaning.monitoring.goToWorkPos )
      wire#w2
      Coil( "Unit1.Em4.ControlNodes".alignTable."step".transition1[481] )
   END_RUNG
   RUNG wire#w1
      Contact( "Unit1.Em4.ControlNodes".alignTable."step".transition1[481] )
   END_RUNG wire#w2
   RUNG wire#w1
      Contact( "Unit1.Em4.ControlNodes".alignTable."step".transition1[481] )
      { S7_Templates := "time_type := Time" } #statTonTime[481].TON(pt := T#1ms, et =>)
      Move(in := #JOB_4_STEP_90, out1 => "Unit1.Em4.ControlNodes".alignTable.sequence.status.nextStep)
   END_RUNG
   // the same network as SCL:
   "Unit1.Em4.ControlNodes".alignTable."step".action1[481] := ("Unit1.Em4.ControlNodes".alignTable.sequence.status.currentStep = #JOB_4_STEP_81) AND "Unit1.Em4.ControlNodes".alignTable.sequence.status.seqActive;
   "Unit1.Em4.ControlNodes".alignTable."step".transition1[481] := ("Unit1.Em4.ControlNodes".alignTable.sequence.status.currentStep = #JOB_4_STEP_81) AND "Unit1.Em4.ControlNodes".alignTable.sequence.status.seqActive AND ("Unit1.Em4.HmiInterface".cmAnodeGlassCleaning.monitoring.goToWorkPos OR "Unit1.Em4.ControlNodes".alignTable."step".transition1[481]);
   #statTonTime[481].TON(IN := ("Unit1.Em4.ControlNodes".alignTable.sequence.status.currentStep = #JOB_4_STEP_81) AND "Unit1.Em4.ControlNodes".alignTable.sequence.status.seqActive AND "Unit1.Em4.ControlNodes".alignTable."step".transition1[481],
                         PT := T#1ms);
   IF #statTonTime[481].Q THEN
       "Unit1.Em4.ControlNodes".alignTable.sequence.status.nextStep := #JOB_4_STEP_90;
   END_IF;
END_REGION

REGION Network 37: Step[490] : JOB[4] Condition
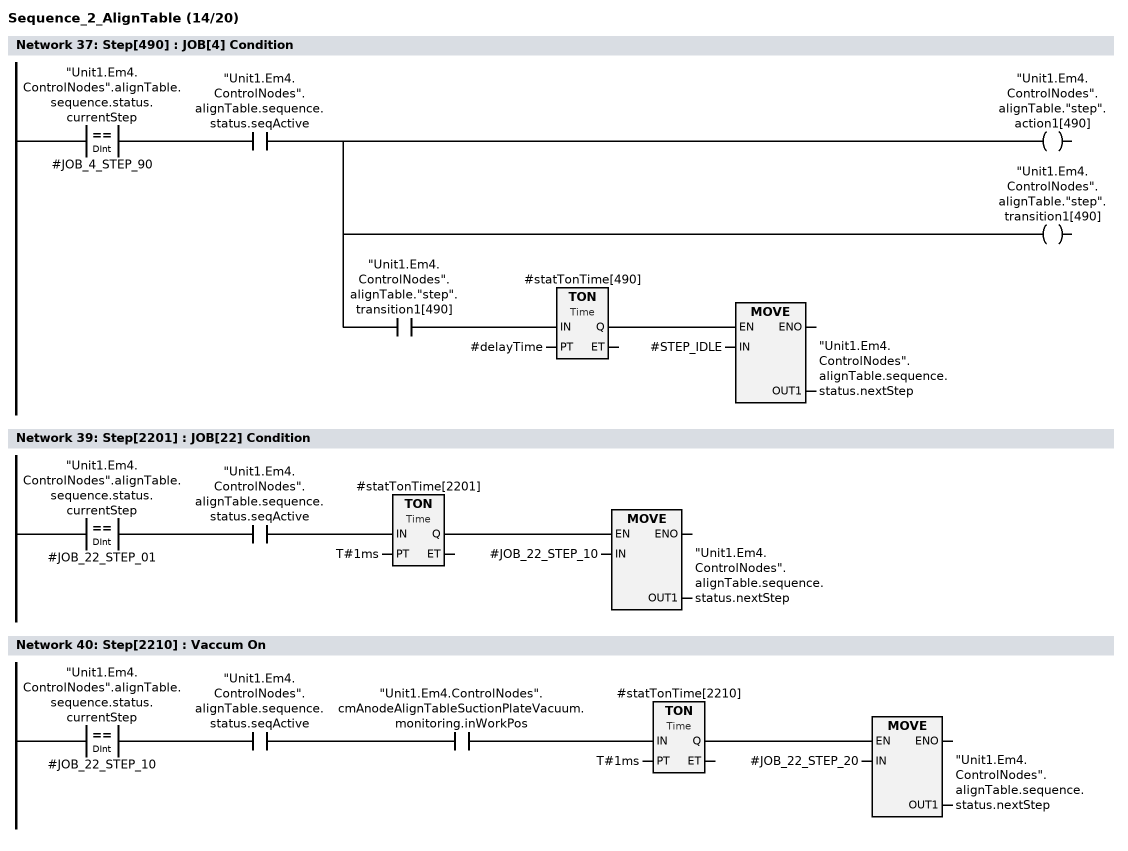
   RUNG wire#powerrail
      { S7_Templates := "SrcType := DInt" } EQ_Contact(in1 := "Unit1.Em4.ControlNodes".alignTable.sequence.status.currentStep, in2 := #JOB_4_STEP_90)
      Contact( "Unit1.Em4.ControlNodes".alignTable.sequence.status.seqActive )
      wire#w1
      Coil( "Unit1.Em4.ControlNodes".alignTable."step".action1[490] )
   END_RUNG
   RUNG wire#w1
      Coil( "Unit1.Em4.ControlNodes".alignTable."step".transition1[490] )
   END_RUNG
   RUNG wire#w1
      Contact( "Unit1.Em4.ControlNodes".alignTable."step".transition1[490] )
      { S7_Templates := "time_type := Time" } #statTonTime[490].TON(pt := #delayTime, et =>)
      Move(in := #STEP_IDLE, out1 => "Unit1.Em4.ControlNodes".alignTable.sequence.status.nextStep)
   END_RUNG
   // the same network as SCL:
   "Unit1.Em4.ControlNodes".alignTable."step".action1[490] := ("Unit1.Em4.ControlNodes".alignTable.sequence.status.currentStep = #JOB_4_STEP_90) AND "Unit1.Em4.ControlNodes".alignTable.sequence.status.seqActive;
   "Unit1.Em4.ControlNodes".alignTable."step".transition1[490] := ("Unit1.Em4.ControlNodes".alignTable.sequence.status.currentStep = #JOB_4_STEP_90) AND "Unit1.Em4.ControlNodes".alignTable.sequence.status.seqActive;
   #statTonTime[490].TON(IN := ("Unit1.Em4.ControlNodes".alignTable.sequence.status.currentStep = #JOB_4_STEP_90) AND "Unit1.Em4.ControlNodes".alignTable.sequence.status.seqActive AND "Unit1.Em4.ControlNodes".alignTable."step".transition1[490],
                         PT := #delayTime);
   IF #statTonTime[490].Q THEN
       "Unit1.Em4.ControlNodes".alignTable.sequence.status.nextStep := #STEP_IDLE;
   END_IF;
END_REGION

REGION Network 38: ******************** JOB[22] Motion ********************
END_REGION

REGION Network 39: Step[2201] : JOB[22] Condition
   RUNG wire#powerrail
      { S7_Templates := "SrcType := DInt" } EQ_Contact(in1 := "Unit1.Em4.ControlNodes".alignTable.sequence.status.currentStep, in2 := #JOB_22_STEP_01)
      Contact( "Unit1.Em4.ControlNodes".alignTable.sequence.status.seqActive )
      { S7_Templates := "time_type := Time" } #statTonTime[2201].TON(pt := T#1ms, et =>)
      Move(in := #JOB_22_STEP_10, out1 => "Unit1.Em4.ControlNodes".alignTable.sequence.status.nextStep)
   END_RUNG
   // the same network as SCL:
   #statTonTime[2201].TON(IN := ("Unit1.Em4.ControlNodes".alignTable.sequence.status.currentStep = #JOB_22_STEP_01) AND "Unit1.Em4.ControlNodes".alignTable.sequence.status.seqActive,
                          PT := T#1ms);
   IF #statTonTime[2201].Q THEN
       "Unit1.Em4.ControlNodes".alignTable.sequence.status.nextStep := #JOB_22_STEP_10;
   END_IF;
END_REGION

REGION Network 40: Step[2210] : Vaccum On
   RUNG wire#powerrail
      { S7_Templates := "SrcType := DInt" } EQ_Contact(in1 := "Unit1.Em4.ControlNodes".alignTable.sequence.status.currentStep, in2 := #JOB_22_STEP_10)
      Contact( "Unit1.Em4.ControlNodes".alignTable.sequence.status.seqActive )
      Contact( "Unit1.Em4.ControlNodes".cmAnodeAlignTableSuctionPlateVacuum.monitoring.inWorkPos )
      { S7_Templates := "time_type := Time" } #statTonTime[2210].TON(pt := T#1ms, et =>)
      Move(in := #JOB_22_STEP_20, out1 => "Unit1.Em4.ControlNodes".alignTable.sequence.status.nextStep)
   END_RUNG
   // the same network as SCL:
   #statTonTime[2210].TON(IN := ("Unit1.Em4.ControlNodes".alignTable.sequence.status.currentStep = #JOB_22_STEP_10) AND "Unit1.Em4.ControlNodes".alignTable.sequence.status.seqActive AND "Unit1.Em4.ControlNodes".cmAnodeAlignTableSuctionPlateVacuum.monitoring.inWorkPos,
                          PT := T#1ms);
   IF #statTonTime[2210].Q THEN
       "Unit1.Em4.ControlNodes".alignTable.sequence.status.nextStep := #JOB_22_STEP_20;
   END_IF;
END_REGION

REGION Network 41: Step[2220] : Vision Start
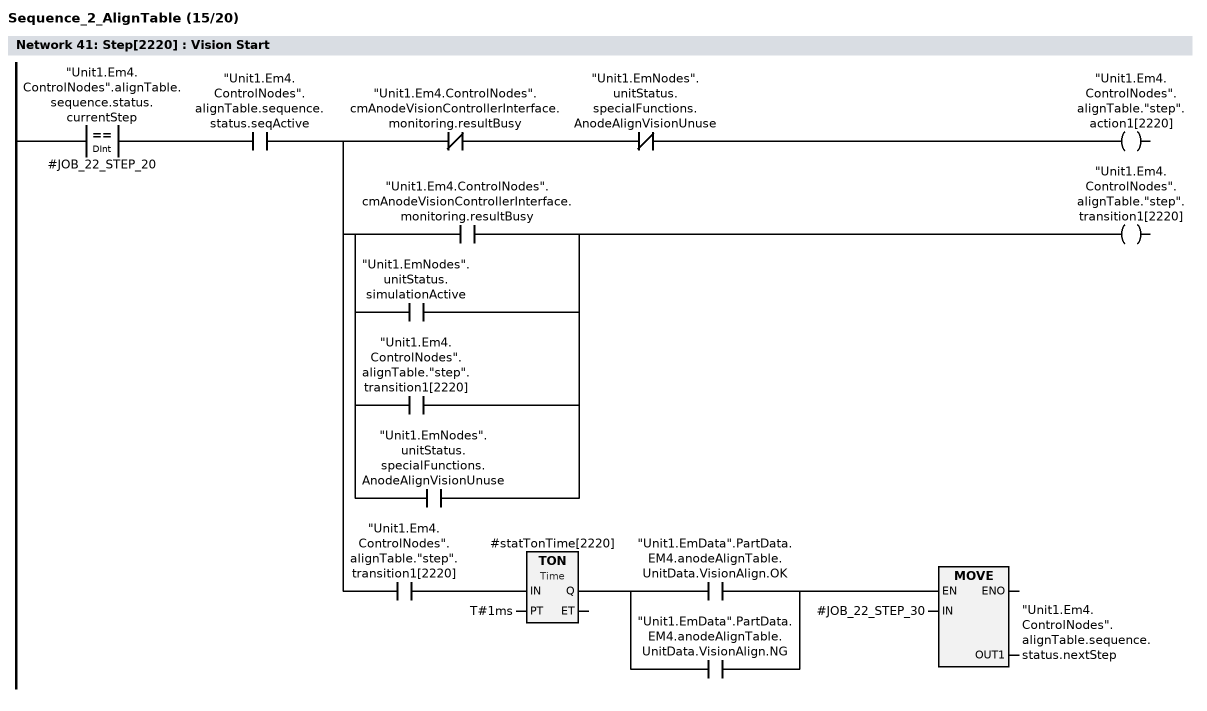
   RUNG wire#powerrail
      { S7_Templates := "SrcType := DInt" } EQ_Contact(in1 := "Unit1.Em4.ControlNodes".alignTable.sequence.status.currentStep, in2 := #JOB_22_STEP_20)
      Contact( "Unit1.Em4.ControlNodes".alignTable.sequence.status.seqActive )
      wire#w1
      I_Contact( "Unit1.Em4.ControlNodes".cmAnodeVisionControllerInterface.monitoring.resultBusy )
      I_Contact( "Unit1.EmNodes".unitStatus.specialFunctions.AnodeAlignVisionUnuse )
      Coil( "Unit1.Em4.ControlNodes".alignTable."step".action1[2220] )
   END_RUNG
   RUNG wire#w1
      Contact( "Unit1.Em4.ControlNodes".cmAnodeVisionControllerInterface.monitoring.resultBusy )
      wire#w2
      Coil( "Unit1.Em4.ControlNodes".alignTable."step".transition1[2220] )
   END_RUNG
   RUNG wire#w1
      Contact( "Unit1.EmNodes".unitStatus.simulationActive )
   END_RUNG wire#w2
   RUNG wire#w1
      Contact( "Unit1.Em4.ControlNodes".alignTable."step".transition1[2220] )
   END_RUNG wire#w2
   RUNG wire#w1
      Contact( "Unit1.EmNodes".unitStatus.specialFunctions.AnodeAlignVisionUnuse )
   END_RUNG wire#w2
   RUNG wire#w1
      Contact( "Unit1.Em4.ControlNodes".alignTable."step".transition1[2220] )
      { S7_Templates := "time_type := Time" } #statTonTime[2220].TON(pt := T#1ms, et =>)
      wire#w3
      Contact( "Unit1.EmData".PartData.EM4.anodeAlignTable.UnitData.VisionAlign.OK )
      wire#w4
      Move(in := #JOB_22_STEP_30, out1 => "Unit1.Em4.ControlNodes".alignTable.sequence.status.nextStep)
   END_RUNG
   RUNG wire#w3
      Contact( "Unit1.EmData".PartData.EM4.anodeAlignTable.UnitData.VisionAlign.NG )
   END_RUNG wire#w4
   // the same network as SCL:
   #_w1 := ("Unit1.Em4.ControlNodes".alignTable.sequence.status.currentStep = #JOB_22_STEP_20) AND "Unit1.Em4.ControlNodes".alignTable.sequence.status.seqActive;
   "Unit1.Em4.ControlNodes".alignTable."step".action1[2220] := #_w1 AND NOT "Unit1.Em4.ControlNodes".cmAnodeVisionControllerInterface.monitoring.resultBusy AND NOT "Unit1.EmNodes".unitStatus.specialFunctions.AnodeAlignVisionUnuse;
   "Unit1.Em4.ControlNodes".alignTable."step".transition1[2220] := #_w1 AND ("Unit1.Em4.ControlNodes".cmAnodeVisionControllerInterface.monitoring.resultBusy OR "Unit1.EmNodes".unitStatus.simulationActive OR "Unit1.Em4.ControlNodes".alignTable."step".transition1[2220] OR "Unit1.EmNodes".unitStatus.specialFunctions.AnodeAlignVisionUnuse);
   #statTonTime[2220].TON(IN := #_w1 AND "Unit1.Em4.ControlNodes".alignTable."step".transition1[2220],
                          PT := T#1ms);
   IF #statTonTime[2220].Q AND ("Unit1.EmData".PartData.EM4.anodeAlignTable.UnitData.VisionAlign.OK OR "Unit1.EmData".PartData.EM4.anodeAlignTable.UnitData.VisionAlign.NG) THEN
       "Unit1.Em4.ControlNodes".alignTable.sequence.status.nextStep := #JOB_22_STEP_30;
   END_IF;
END_REGION

REGION Network 42: Step[2230] : Vision Result
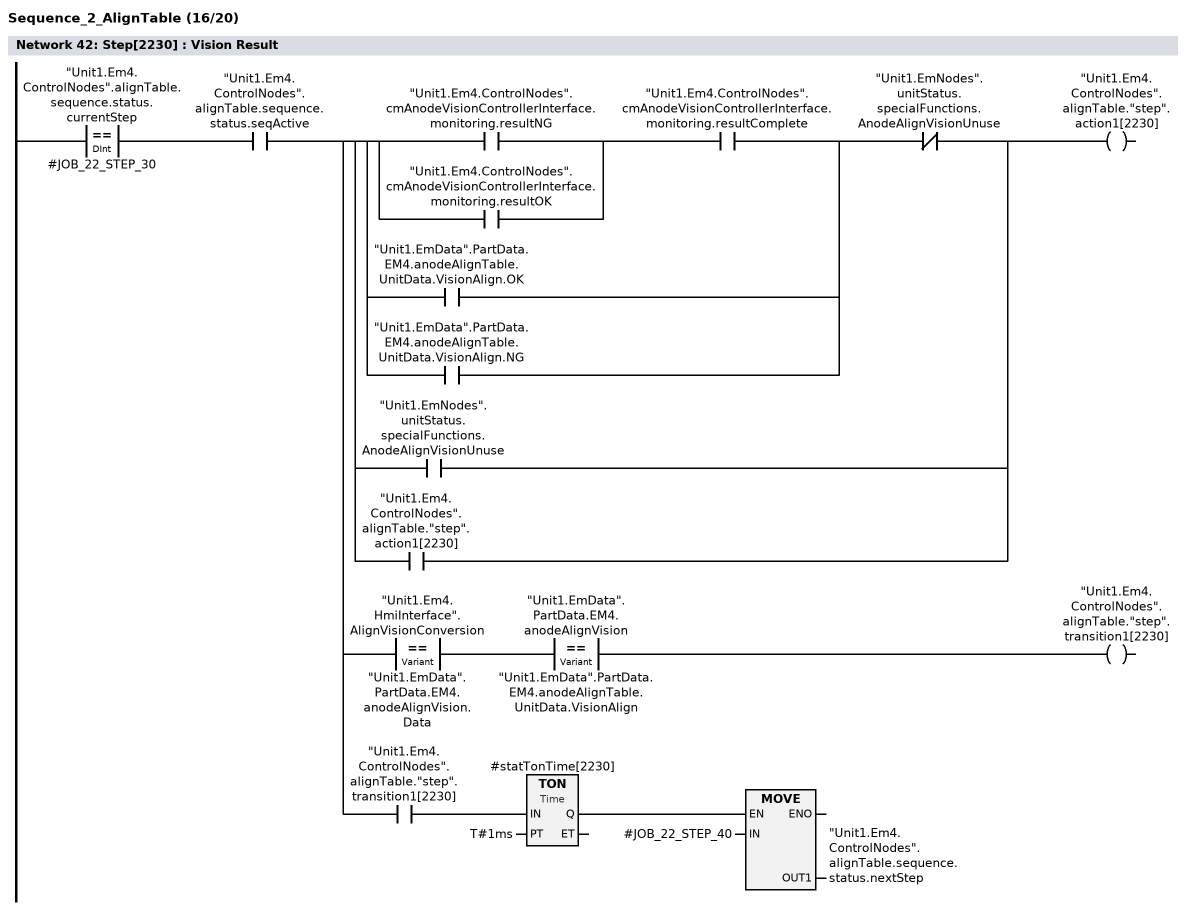
   RUNG wire#powerrail
      { S7_Templates := "SrcType := DInt" } EQ_Contact(in1 := "Unit1.Em4.ControlNodes".alignTable.sequence.status.currentStep, in2 := #JOB_22_STEP_30)
      Contact( "Unit1.Em4.ControlNodes".alignTable.sequence.status.seqActive )
      wire#w1
      Contact( "Unit1.Em4.ControlNodes".cmAnodeVisionControllerInterface.monitoring.resultNG )
      wire#w2
      Contact( "Unit1.Em4.ControlNodes".cmAnodeVisionControllerInterface.monitoring.resultComplete )
      wire#w3
      I_Contact( "Unit1.EmNodes".unitStatus.specialFunctions.AnodeAlignVisionUnuse )
      wire#w4
      Coil( "Unit1.Em4.ControlNodes".alignTable."step".action1[2230] )
   END_RUNG
   RUNG wire#w1
      Contact( "Unit1.Em4.ControlNodes".cmAnodeVisionControllerInterface.monitoring.resultOK )
   END_RUNG wire#w2
   RUNG wire#w1
      Contact( "Unit1.EmData".PartData.EM4.anodeAlignTable.UnitData.VisionAlign.OK )
   END_RUNG wire#w3
   RUNG wire#w1
      Contact( "Unit1.EmData".PartData.EM4.anodeAlignTable.UnitData.VisionAlign.NG )
   END_RUNG wire#w3
   RUNG wire#w1
      Contact( "Unit1.EmNodes".unitStatus.specialFunctions.AnodeAlignVisionUnuse )
   END_RUNG wire#w4
   RUNG wire#w1
      Contact( "Unit1.Em4.ControlNodes".alignTable."step".action1[2230] )
   END_RUNG wire#w4
   RUNG wire#w1
      { S7_Templates := "SrcType := Variant" } EQ_Contact(in1 := "Unit1.Em4.HmiInterface".AlignVisionConversion, in2 := "Unit1.EmData".PartData.EM4.anodeAlignVision.Data)
      { S7_Templates := "SrcType := Variant" } EQ_Contact(in1 := "Unit1.EmData".PartData.EM4.anodeAlignVision, in2 := "Unit1.EmData".PartData.EM4.anodeAlignTable.UnitData.VisionAlign)
      Coil( "Unit1.Em4.ControlNodes".alignTable."step".transition1[2230] )
   END_RUNG
   RUNG wire#w1
      Contact( "Unit1.Em4.ControlNodes".alignTable."step".transition1[2230] )
      { S7_Templates := "time_type := Time" } #statTonTime[2230].TON(pt := T#1ms, et =>)
      Move(in := #JOB_22_STEP_40, out1 => "Unit1.Em4.ControlNodes".alignTable.sequence.status.nextStep)
   END_RUNG
   // the same network as SCL:
   #_w1 := ("Unit1.Em4.ControlNodes".alignTable.sequence.status.currentStep = #JOB_22_STEP_30) AND "Unit1.Em4.ControlNodes".alignTable.sequence.status.seqActive;
   "Unit1.Em4.ControlNodes".alignTable."step".action1[2230] := #_w1 AND ((((("Unit1.Em4.ControlNodes".cmAnodeVisionControllerInterface.monitoring.resultNG OR "Unit1.Em4.ControlNodes".cmAnodeVisionControllerInterface.monitoring.resultOK) AND "Unit1.Em4.ControlNodes".cmAnodeVisionControllerInterface.monitoring.resultComplete) OR "Unit1.EmData".PartData.EM4.anodeAlignTable.UnitData.VisionAlign.OK OR "Unit1.EmData".PartData.EM4.anodeAlignTable.UnitData.VisionAlign.NG) AND NOT "Unit1.EmNodes".unitStatus.specialFunctions.AnodeAlignVisionUnuse) OR "Unit1.EmNodes".unitStatus.specialFunctions.AnodeAlignVisionUnuse OR "Unit1.Em4.ControlNodes".alignTable."step".action1[2230]);
   "Unit1.Em4.ControlNodes".alignTable."step".transition1[2230] := #_w1 AND ("Unit1.Em4.HmiInterface".AlignVisionConversion = "Unit1.EmData".PartData.EM4.anodeAlignVision.Data) AND ("Unit1.EmData".PartData.EM4.anodeAlignVision = "Unit1.EmData".PartData.EM4.anodeAlignTable.UnitData.VisionAlign);
   #statTonTime[2230].TON(IN := #_w1 AND "Unit1.Em4.ControlNodes".alignTable."step".transition1[2230],
                          PT := T#1ms);
   IF #statTonTime[2230].Q THEN
       "Unit1.Em4.ControlNodes".alignTable.sequence.status.nextStep := #JOB_22_STEP_40;
   END_IF;
END_REGION

REGION Network 43: Step[2240] : Align Table X,Y1,Y2-Axis Work Pos
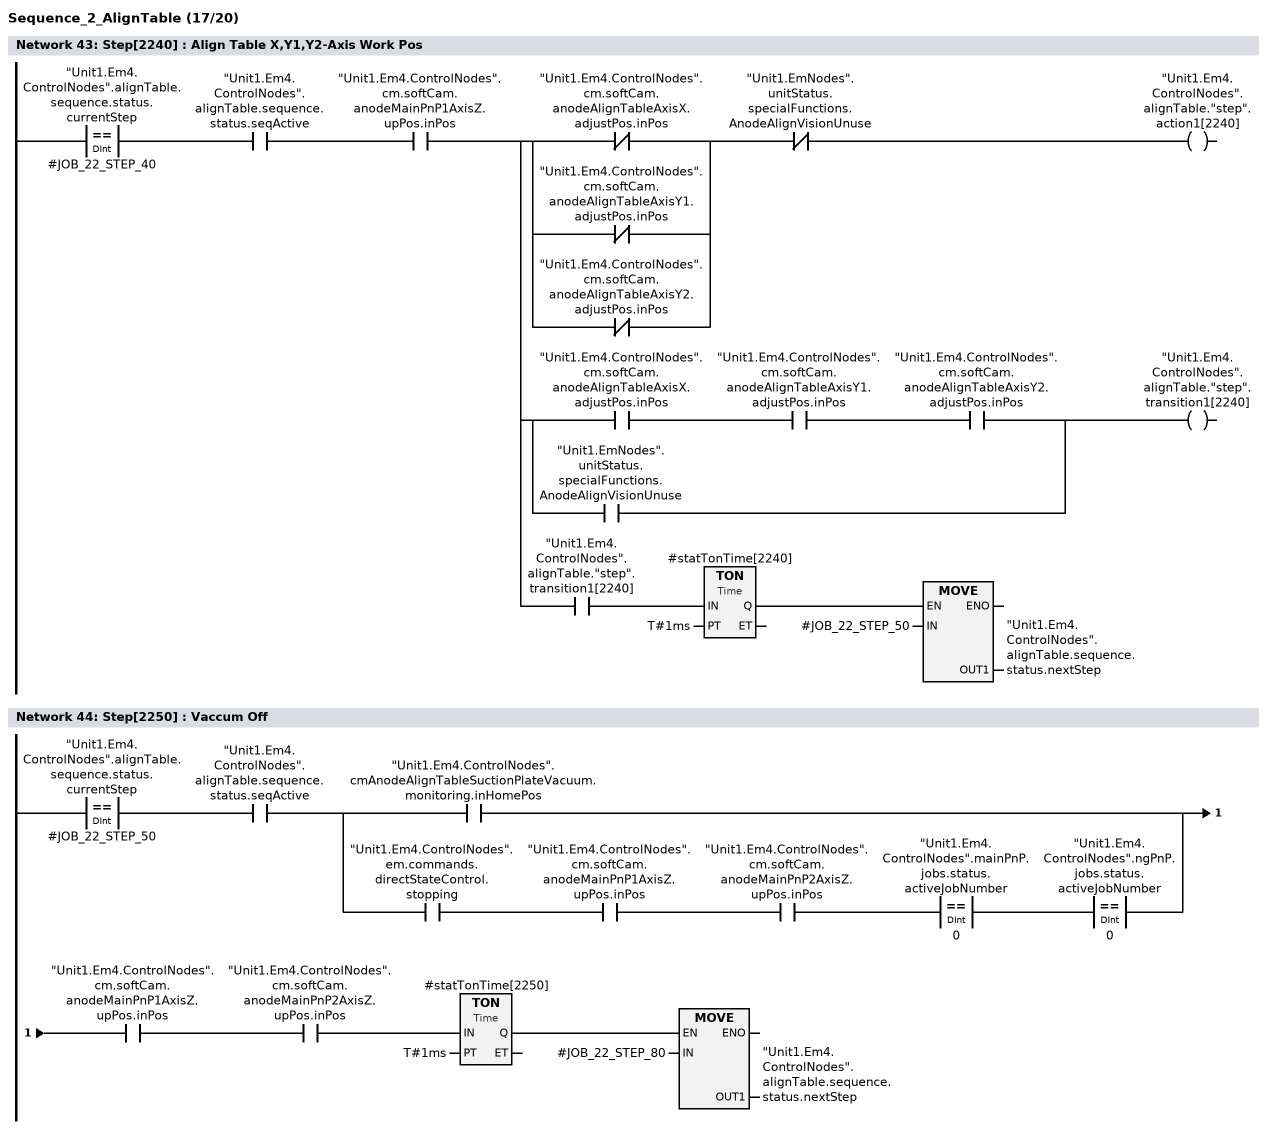
   RUNG wire#powerrail
      { S7_Templates := "SrcType := DInt" } EQ_Contact(in1 := "Unit1.Em4.ControlNodes".alignTable.sequence.status.currentStep, in2 := #JOB_22_STEP_40)
      Contact( "Unit1.Em4.ControlNodes".alignTable.sequence.status.seqActive )
      Contact( "Unit1.Em4.ControlNodes".cm.softCam.anodeMainPnP1AxisZ.upPos.inPos )
      wire#w1
      I_Contact( "Unit1.Em4.ControlNodes".cm.softCam.anodeAlignTableAxisX.adjustPos.inPos )
      wire#w2
      I_Contact( "Unit1.EmNodes".unitStatus.specialFunctions.AnodeAlignVisionUnuse )
      Coil( "Unit1.Em4.ControlNodes".alignTable."step".action1[2240] )
   END_RUNG
   RUNG wire#w1
      I_Contact( "Unit1.Em4.ControlNodes".cm.softCam.anodeAlignTableAxisY1.adjustPos.inPos )
   END_RUNG wire#w2
   RUNG wire#w1
      I_Contact( "Unit1.Em4.ControlNodes".cm.softCam.anodeAlignTableAxisY2.adjustPos.inPos )
   END_RUNG wire#w2
   RUNG wire#w1
      Contact( "Unit1.Em4.ControlNodes".cm.softCam.anodeAlignTableAxisX.adjustPos.inPos )
      Contact( "Unit1.Em4.ControlNodes".cm.softCam.anodeAlignTableAxisY1.adjustPos.inPos )
      Contact( "Unit1.Em4.ControlNodes".cm.softCam.anodeAlignTableAxisY2.adjustPos.inPos )
      wire#w3
      Coil( "Unit1.Em4.ControlNodes".alignTable."step".transition1[2240] )
   END_RUNG
   RUNG wire#w1
      Contact( "Unit1.EmNodes".unitStatus.specialFunctions.AnodeAlignVisionUnuse )
   END_RUNG wire#w3
   RUNG wire#w1
      Contact( "Unit1.Em4.ControlNodes".alignTable."step".transition1[2240] )
      { S7_Templates := "time_type := Time" } #statTonTime[2240].TON(pt := T#1ms, et =>)
      Move(in := #JOB_22_STEP_50, out1 => "Unit1.Em4.ControlNodes".alignTable.sequence.status.nextStep)
   END_RUNG
   // the same network as SCL:
   #_w1 := ("Unit1.Em4.ControlNodes".alignTable.sequence.status.currentStep = #JOB_22_STEP_40) AND "Unit1.Em4.ControlNodes".alignTable.sequence.status.seqActive AND "Unit1.Em4.ControlNodes".cm.softCam.anodeMainPnP1AxisZ.upPos.inPos;
   "Unit1.Em4.ControlNodes".alignTable."step".action1[2240] := #_w1 AND (NOT "Unit1.Em4.ControlNodes".cm.softCam.anodeAlignTableAxisX.adjustPos.inPos OR NOT "Unit1.Em4.ControlNodes".cm.softCam.anodeAlignTableAxisY1.adjustPos.inPos OR NOT "Unit1.Em4.ControlNodes".cm.softCam.anodeAlignTableAxisY2.adjustPos.inPos) AND NOT "Unit1.EmNodes".unitStatus.specialFunctions.AnodeAlignVisionUnuse;
   "Unit1.Em4.ControlNodes".alignTable."step".transition1[2240] := #_w1 AND (("Unit1.Em4.ControlNodes".cm.softCam.anodeAlignTableAxisX.adjustPos.inPos AND "Unit1.Em4.ControlNodes".cm.softCam.anodeAlignTableAxisY1.adjustPos.inPos AND "Unit1.Em4.ControlNodes".cm.softCam.anodeAlignTableAxisY2.adjustPos.inPos) OR "Unit1.EmNodes".unitStatus.specialFunctions.AnodeAlignVisionUnuse);
   #statTonTime[2240].TON(IN := #_w1 AND "Unit1.Em4.ControlNodes".alignTable."step".transition1[2240],
                          PT := T#1ms);
   IF #statTonTime[2240].Q THEN
       "Unit1.Em4.ControlNodes".alignTable.sequence.status.nextStep := #JOB_22_STEP_50;
   END_IF;
END_REGION

REGION Network 44: Step[2250] : Vaccum Off
   RUNG wire#powerrail
      { S7_Templates := "SrcType := DInt" } EQ_Contact(in1 := "Unit1.Em4.ControlNodes".alignTable.sequence.status.currentStep, in2 := #JOB_22_STEP_50)
      Contact( "Unit1.Em4.ControlNodes".alignTable.sequence.status.seqActive )
      wire#w1
      Contact( "Unit1.Em4.ControlNodes".cmAnodeAlignTableSuctionPlateVacuum.monitoring.inHomePos )
      wire#w2
      Contact( "Unit1.Em4.ControlNodes".cm.softCam.anodeMainPnP1AxisZ.upPos.inPos )
      Contact( "Unit1.Em4.ControlNodes".cm.softCam.anodeMainPnP2AxisZ.upPos.inPos )
      { S7_Templates := "time_type := Time" } #statTonTime[2250].TON(pt := T#1ms, et =>)
      Move(in := #JOB_22_STEP_80, out1 => "Unit1.Em4.ControlNodes".alignTable.sequence.status.nextStep)
   END_RUNG
   RUNG wire#w1
      Contact( "Unit1.Em4.ControlNodes".em.commands.directStateControl.stopping )
      Contact( "Unit1.Em4.ControlNodes".cm.softCam.anodeMainPnP1AxisZ.upPos.inPos )
      Contact( "Unit1.Em4.ControlNodes".cm.softCam.anodeMainPnP2AxisZ.upPos.inPos )
      { S7_Templates := "SrcType := DInt" } EQ_Contact(in1 := "Unit1.Em4.ControlNodes".mainPnP.jobs.status.activeJobNumber, in2 := 0)
      { S7_Templates := "SrcType := DInt" } EQ_Contact(in1 := "Unit1.Em4.ControlNodes".ngPnP.jobs.status.activeJobNumber, in2 := 0)
   END_RUNG wire#w2
   // the same network as SCL:
   #statTonTime[2250].TON(IN := ("Unit1.Em4.ControlNodes".alignTable.sequence.status.currentStep = #JOB_22_STEP_50) AND "Unit1.Em4.ControlNodes".alignTable.sequence.status.seqActive AND ("Unit1.Em4.ControlNodes".cmAnodeAlignTableSuctionPlateVacuum.monitoring.inHomePos OR ("Unit1.Em4.ControlNodes".em.commands.directStateControl.stopping AND "Unit1.Em4.ControlNodes".cm.softCam.anodeMainPnP1AxisZ.upPos.inPos AND "Unit1.Em4.ControlNodes".cm.softCam.anodeMainPnP2AxisZ.upPos.inPos AND ("Unit1.Em4.ControlNodes".mainPnP.jobs.status.activeJobNumber = 0) AND ("Unit1.Em4.ControlNodes".ngPnP.jobs.status.activeJobNumber = 0))) AND "Unit1.Em4.ControlNodes".cm.softCam.anodeMainPnP1AxisZ.upPos.inPos AND "Unit1.Em4.ControlNodes".cm.softCam.anodeMainPnP2AxisZ.upPos.inPos,
                          PT := T#1ms);
   IF #statTonTime[2250].Q THEN
       "Unit1.Em4.ControlNodes".alignTable.sequence.status.nextStep := #JOB_22_STEP_80;
   END_IF;
END_REGION

REGION Network 45: Step[2280] : Align Table X,Y1,Y2-Axis Wait Pos
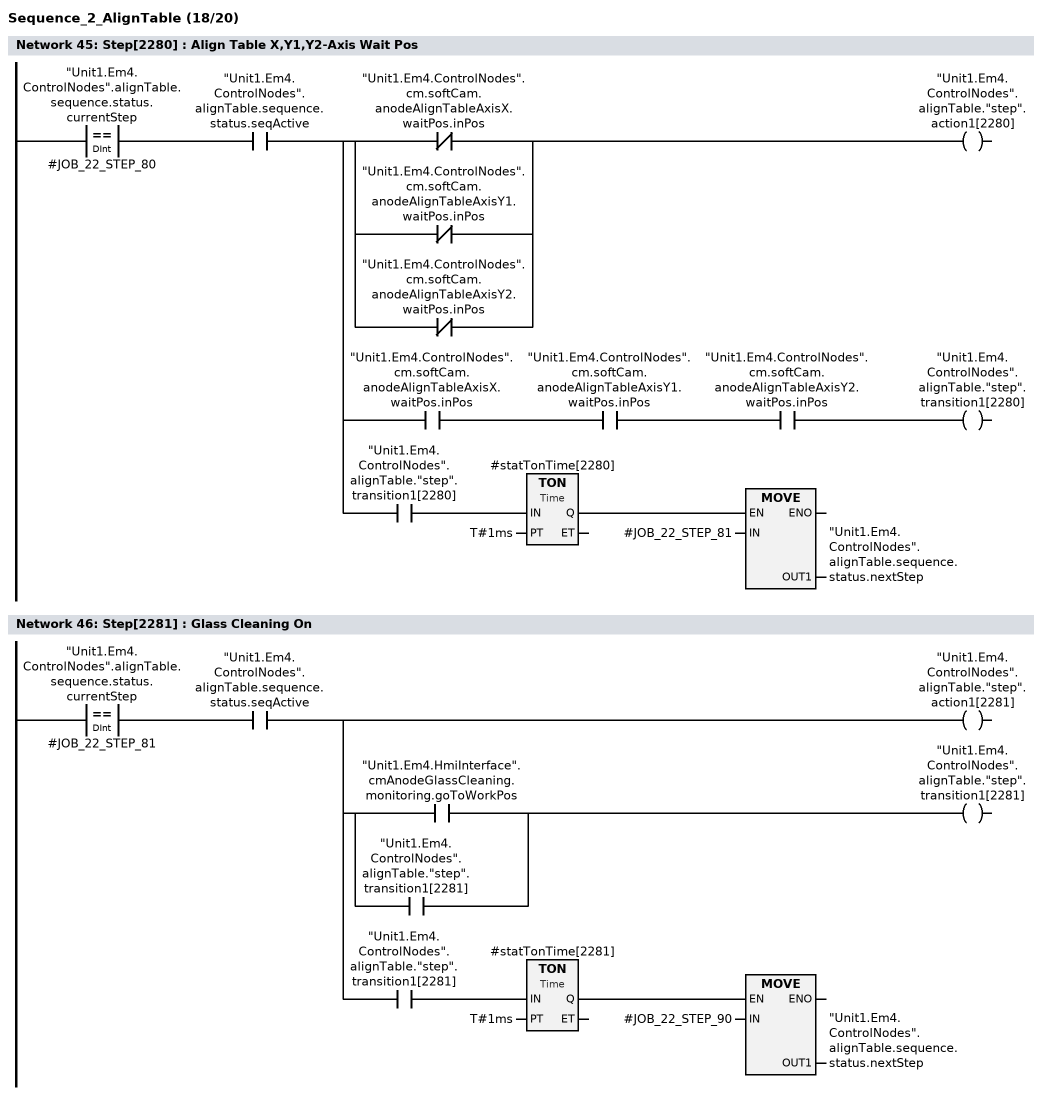
   RUNG wire#powerrail
      { S7_Templates := "SrcType := DInt" } EQ_Contact(in1 := "Unit1.Em4.ControlNodes".alignTable.sequence.status.currentStep, in2 := #JOB_22_STEP_80)
      Contact( "Unit1.Em4.ControlNodes".alignTable.sequence.status.seqActive )
      wire#w1
      I_Contact( "Unit1.Em4.ControlNodes".cm.softCam.anodeAlignTableAxisX.waitPos.inPos )
      wire#w2
      Coil( "Unit1.Em4.ControlNodes".alignTable."step".action1[2280] )
   END_RUNG
   RUNG wire#w1
      I_Contact( "Unit1.Em4.ControlNodes".cm.softCam.anodeAlignTableAxisY1.waitPos.inPos )
   END_RUNG wire#w2
   RUNG wire#w1
      I_Contact( "Unit1.Em4.ControlNodes".cm.softCam.anodeAlignTableAxisY2.waitPos.inPos )
   END_RUNG wire#w2
   RUNG wire#w1
      Contact( "Unit1.Em4.ControlNodes".cm.softCam.anodeAlignTableAxisX.waitPos.inPos )
      Contact( "Unit1.Em4.ControlNodes".cm.softCam.anodeAlignTableAxisY1.waitPos.inPos )
      Contact( "Unit1.Em4.ControlNodes".cm.softCam.anodeAlignTableAxisY2.waitPos.inPos )
      Coil( "Unit1.Em4.ControlNodes".alignTable."step".transition1[2280] )
   END_RUNG
   RUNG wire#w1
      Contact( "Unit1.Em4.ControlNodes".alignTable."step".transition1[2280] )
      { S7_Templates := "time_type := Time" } #statTonTime[2280].TON(pt := T#1ms, et =>)
      Move(in := #JOB_22_STEP_81, out1 => "Unit1.Em4.ControlNodes".alignTable.sequence.status.nextStep)
   END_RUNG
   // the same network as SCL:
   #_w1 := ("Unit1.Em4.ControlNodes".alignTable.sequence.status.currentStep = #JOB_22_STEP_80) AND "Unit1.Em4.ControlNodes".alignTable.sequence.status.seqActive;
   "Unit1.Em4.ControlNodes".alignTable."step".action1[2280] := #_w1 AND (NOT "Unit1.Em4.ControlNodes".cm.softCam.anodeAlignTableAxisX.waitPos.inPos OR NOT "Unit1.Em4.ControlNodes".cm.softCam.anodeAlignTableAxisY1.waitPos.inPos OR NOT "Unit1.Em4.ControlNodes".cm.softCam.anodeAlignTableAxisY2.waitPos.inPos);
   "Unit1.Em4.ControlNodes".alignTable."step".transition1[2280] := #_w1 AND "Unit1.Em4.ControlNodes".cm.softCam.anodeAlignTableAxisX.waitPos.inPos AND "Unit1.Em4.ControlNodes".cm.softCam.anodeAlignTableAxisY1.waitPos.inPos AND "Unit1.Em4.ControlNodes".cm.softCam.anodeAlignTableAxisY2.waitPos.inPos;
   #statTonTime[2280].TON(IN := #_w1 AND "Unit1.Em4.ControlNodes".alignTable."step".transition1[2280],
                          PT := T#1ms);
   IF #statTonTime[2280].Q THEN
       "Unit1.Em4.ControlNodes".alignTable.sequence.status.nextStep := #JOB_22_STEP_81;
   END_IF;
END_REGION

REGION Network 46: Step[2281] : Glass Cleaning On
   RUNG wire#powerrail
      { S7_Templates := "SrcType := DInt" } EQ_Contact(in1 := "Unit1.Em4.ControlNodes".alignTable.sequence.status.currentStep, in2 := #JOB_22_STEP_81)
      Contact( "Unit1.Em4.ControlNodes".alignTable.sequence.status.seqActive )
      wire#w1
      Coil( "Unit1.Em4.ControlNodes".alignTable."step".action1[2281] )
   END_RUNG
   RUNG wire#w1
      Contact( "Unit1.Em4.HmiInterface".cmAnodeGlassCleaning.monitoring.goToWorkPos )
      wire#w2
      Coil( "Unit1.Em4.ControlNodes".alignTable."step".transition1[2281] )
   END_RUNG
   RUNG wire#w1
      Contact( "Unit1.Em4.ControlNodes".alignTable."step".transition1[2281] )
   END_RUNG wire#w2
   RUNG wire#w1
      Contact( "Unit1.Em4.ControlNodes".alignTable."step".transition1[2281] )
      { S7_Templates := "time_type := Time" } #statTonTime[2281].TON(pt := T#1ms, et =>)
      Move(in := #JOB_22_STEP_90, out1 => "Unit1.Em4.ControlNodes".alignTable.sequence.status.nextStep)
   END_RUNG
   // the same network as SCL:
   "Unit1.Em4.ControlNodes".alignTable."step".action1[2281] := ("Unit1.Em4.ControlNodes".alignTable.sequence.status.currentStep = #JOB_22_STEP_81) AND "Unit1.Em4.ControlNodes".alignTable.sequence.status.seqActive;
   "Unit1.Em4.ControlNodes".alignTable."step".transition1[2281] := ("Unit1.Em4.ControlNodes".alignTable.sequence.status.currentStep = #JOB_22_STEP_81) AND "Unit1.Em4.ControlNodes".alignTable.sequence.status.seqActive AND ("Unit1.Em4.HmiInterface".cmAnodeGlassCleaning.monitoring.goToWorkPos OR "Unit1.Em4.ControlNodes".alignTable."step".transition1[2281]);
   #statTonTime[2281].TON(IN := ("Unit1.Em4.ControlNodes".alignTable.sequence.status.currentStep = #JOB_22_STEP_81) AND "Unit1.Em4.ControlNodes".alignTable.sequence.status.seqActive AND "Unit1.Em4.ControlNodes".alignTable."step".transition1[2281],
                          PT := T#1ms);
   IF #statTonTime[2281].Q THEN
       "Unit1.Em4.ControlNodes".alignTable.sequence.status.nextStep := #JOB_22_STEP_90;
   END_IF;
END_REGION

REGION Network 47: Step[2290] : JOB[22] Condition
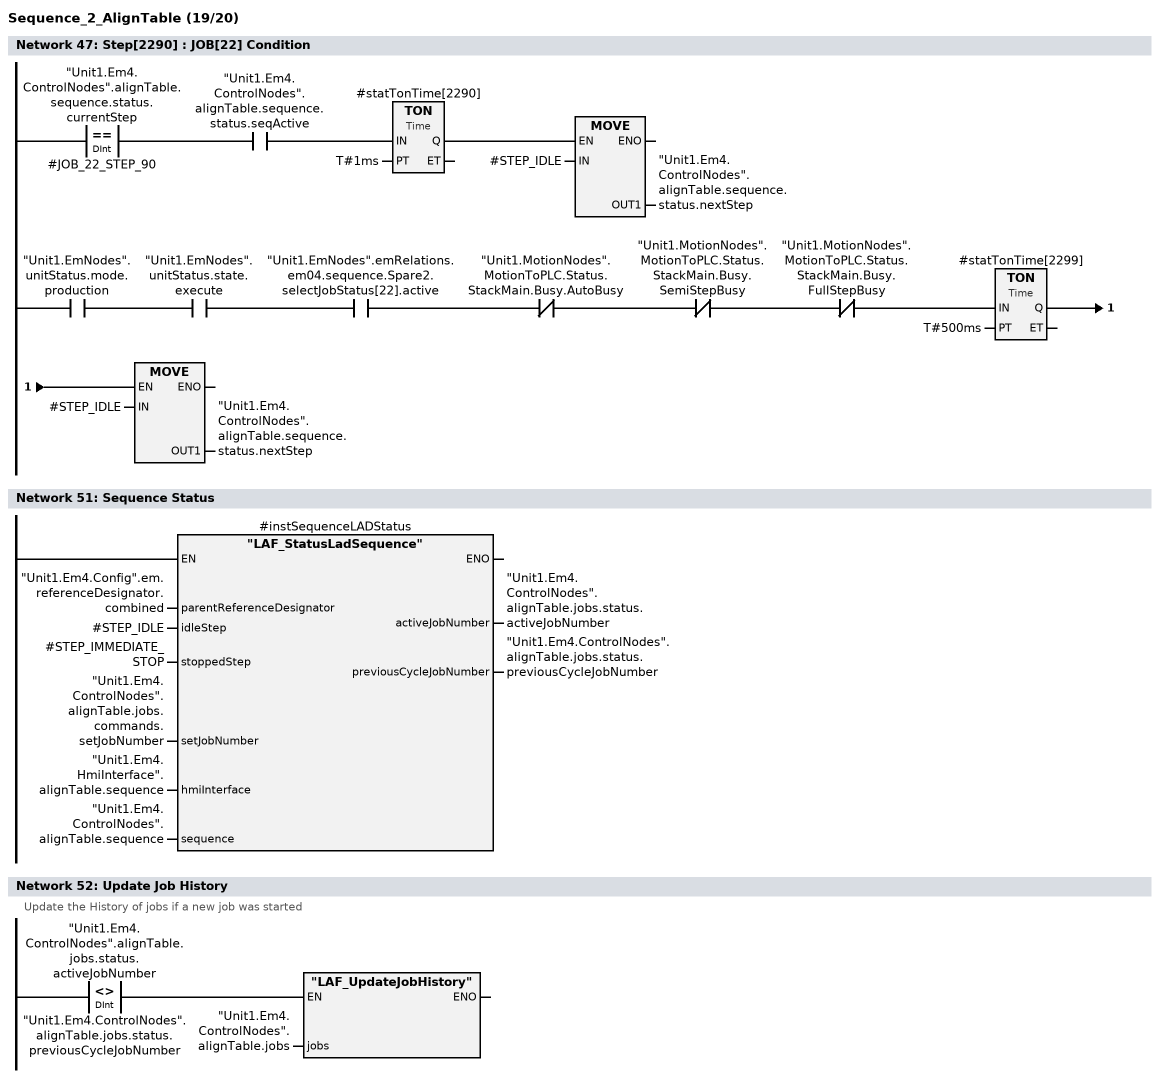
   RUNG wire#powerrail
      { S7_Templates := "SrcType := DInt" } EQ_Contact(in1 := "Unit1.Em4.ControlNodes".alignTable.sequence.status.currentStep, in2 := #JOB_22_STEP_90)
      Contact( "Unit1.Em4.ControlNodes".alignTable.sequence.status.seqActive )
      { S7_Templates := "time_type := Time" } #statTonTime[2290].TON(pt := T#1ms, et =>)
      Move(in := #STEP_IDLE, out1 => "Unit1.Em4.ControlNodes".alignTable.sequence.status.nextStep)
   END_RUNG
   RUNG wire#powerrail
      Contact( "Unit1.EmNodes".unitStatus.mode.production )
      Contact( "Unit1.EmNodes".unitStatus.state.execute )
      Contact( "Unit1.EmNodes".emRelations.em04.sequence.Spare2.selectJobStatus[22].active )
      I_Contact( "Unit1.MotionNodes".MotionToPLC.Status.StackMain.Busy.AutoBusy )
      I_Contact( "Unit1.MotionNodes".MotionToPLC.Status.StackMain.Busy.SemiStepBusy )
      I_Contact( "Unit1.MotionNodes".MotionToPLC.Status.StackMain.Busy.FullStepBusy )
      { S7_Templates := "time_type := Time" } #statTonTime[2299].TON(pt := T#500ms, et =>)
      Move(in := #STEP_IDLE, out1 => "Unit1.Em4.ControlNodes".alignTable.sequence.status.nextStep)
   END_RUNG
   // the same network as SCL:
   #statTonTime[2290].TON(IN := ("Unit1.Em4.ControlNodes".alignTable.sequence.status.currentStep = #JOB_22_STEP_90) AND "Unit1.Em4.ControlNodes".alignTable.sequence.status.seqActive,
                          PT := T#1ms);
   IF #statTonTime[2290].Q THEN
       "Unit1.Em4.ControlNodes".alignTable.sequence.status.nextStep := #STEP_IDLE;
   END_IF;
   #statTonTime[2299].TON(IN := "Unit1.EmNodes".unitStatus.mode.production AND "Unit1.EmNodes".unitStatus.state.execute AND "Unit1.EmNodes".emRelations.em04.sequence.Spare2.selectJobStatus[22].active AND NOT "Unit1.MotionNodes".MotionToPLC.Status.StackMain.Busy.AutoBusy AND NOT "Unit1.MotionNodes".MotionToPLC.Status.StackMain.Busy.SemiStepBusy AND NOT "Unit1.MotionNodes".MotionToPLC.Status.StackMain.Busy.FullStepBusy,
                          PT := T#500ms);
   IF #statTonTime[2299].Q THEN
       "Unit1.Em4.ControlNodes".alignTable.sequence.status.nextStep := #STEP_IDLE;
   END_IF;
END_REGION

REGION Network 48: *************** IMMEDIATE STOP **************************
END_REGION

REGION Network 49: Immediate Stop
END_REGION

REGION Network 50: *************** Status updates **************************
END_REGION

REGION Network 51: Sequence Status
   RUNG wire#powerrail
      #instSequenceLADStatus(parentReferenceDesignator := "Unit1.Em4.Config".em.referenceDesignator.combined, idleStep := #STEP_IDLE, stoppedStep := #STEP_IMMEDIATE_STOP, setJobNumber := "Unit1.Em4.ControlNodes".alignTable.jobs.commands.setJobNumber, hmiInterface := "Unit1.Em4.HmiInterface".alignTable.sequence, sequence := "Unit1.Em4.ControlNodes".alignTable.sequence, activeJobNumber => "Unit1.Em4.ControlNodes".alignTable.jobs.status.activeJobNumber, previousCycleJobNumber => "Unit1.Em4.ControlNodes".alignTable.jobs.status.previousCycleJobNumber)
   END_RUNG
   // the same network as SCL:
   #instSequenceLADStatus(parentReferenceDesignator := "Unit1.Em4.Config".em.referenceDesignator.combined,   // "LAF_StatusLadSequence"
                          idleStep := #STEP_IDLE,
                          stoppedStep := #STEP_IMMEDIATE_STOP,
                          setJobNumber := "Unit1.Em4.ControlNodes".alignTable.jobs.commands.setJobNumber,
                          hmiInterface := "Unit1.Em4.HmiInterface".alignTable.sequence,
                          sequence := "Unit1.Em4.ControlNodes".alignTable.sequence,
                          activeJobNumber => "Unit1.Em4.ControlNodes".alignTable.jobs.status.activeJobNumber,
                          previousCycleJobNumber => "Unit1.Em4.ControlNodes".alignTable.jobs.status.previousCycleJobNumber);
END_REGION

REGION Network 52: Update Job History
   // Update the History of jobs if a new job was started
   RUNG wire#powerrail
      { S7_Templates := "SrcType := DInt" } NE_Contact(in1 := "Unit1.Em4.ControlNodes".alignTable.jobs.status.activeJobNumber, in2 := "Unit1.Em4.ControlNodes".alignTable.jobs.status.previousCycleJobNumber)
      "LAF_UpdateJobHistory"(jobs := "Unit1.Em4.ControlNodes".alignTable.jobs)
   END_RUNG
   // the same network as SCL:
   IF "Unit1.Em4.ControlNodes".alignTable.jobs.status.activeJobNumber <> "Unit1.Em4.ControlNodes".alignTable.jobs.status.previousCycleJobNumber THEN
       "LAF_UpdateJobHistory"(jobs := "Unit1.Em4.ControlNodes".alignTable.jobs);
   END_IF;
END_REGION

REGION Network 53: Output steps as String
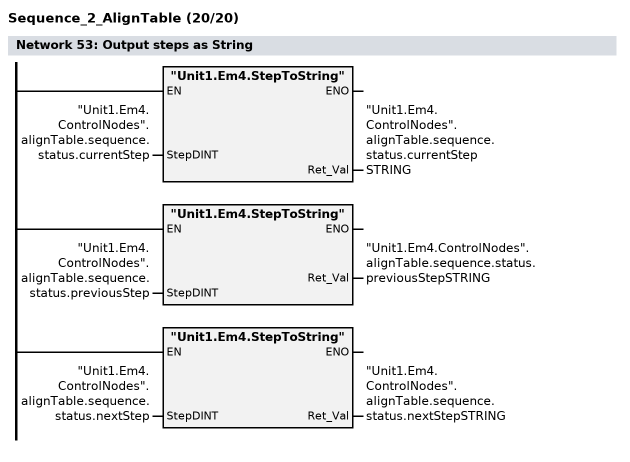
   RUNG wire#powerrail
      "Unit1.Em4.StepToString"(StepDINT := "Unit1.Em4.ControlNodes".alignTable.sequence.status.currentStep, Ret_Val => "Unit1.Em4.ControlNodes".alignTable.sequence.status.currentStepSTRING)
   END_RUNG
   RUNG wire#powerrail
      "Unit1.Em4.StepToString"(StepDINT := "Unit1.Em4.ControlNodes".alignTable.sequence.status.previousStep, Ret_Val => "Unit1.Em4.ControlNodes".alignTable.sequence.status.previousStepSTRING)
   END_RUNG
   RUNG wire#powerrail
      "Unit1.Em4.StepToString"(StepDINT := "Unit1.Em4.ControlNodes".alignTable.sequence.status.nextStep, Ret_Val => "Unit1.Em4.ControlNodes".alignTable.sequence.status.nextStepSTRING)
   END_RUNG
   // the same network as SCL:
   "Unit1.Em4.ControlNodes".alignTable.sequence.status.currentStepSTRING := "Unit1.Em4.StepToString"(StepDINT := "Unit1.Em4.ControlNodes".alignTable.sequence.status.currentStep);
   "Unit1.Em4.ControlNodes".alignTable.sequence.status.previousStepSTRING := "Unit1.Em4.StepToString"(StepDINT := "Unit1.Em4.ControlNodes".alignTable.sequence.status.previousStep);
   "Unit1.Em4.ControlNodes".alignTable.sequence.status.nextStepSTRING := "Unit1.Em4.StepToString"(StepDINT := "Unit1.Em4.ControlNodes".alignTable.sequence.status.nextStep);
END_REGION
END_FUNCTION_BLOCK
